LIN {X 0,Y 418.25,Z 348.011,A -85,B 0,C 180,E1 -10113.677,E2 -10113.677} C_VEL
LIN {X 0,Y 418.241,Z 348.013,A -85,B 0,C 180,E1 -10117.224,E2 -10117.224} C_VEL
LIN {X 0,Y 418.253,Z 348.011,A -85,B 0,C 180,E1 -10119.681,E2 -10119.681} C_VEL
LIN {X 0,Y 418.231,Z 348.014,A -85,B 0,C 180,E1 -10122.321,E2 -10122.321} C_VEL
LIN {X 0,Y 418.241,Z 348.014,A -85,B 0,C 180,E1 -10125.109,E2 -10125.109} C_VEL
LIN {X 0,Y 418.244,Z 348.011,A -85,B 0,C 180,E1 -10127.767,E2 -10127.767} C_VEL
LIN {X 0,Y 418.259,Z 348.01,A -85,B 0,C 180,E1 -10130.618,E2 -10130.618} C_VEL
LIN {X 0,Y 418.245,Z 348.013,A -85,B 0,C 180,E1 -10133.976,E2 -10133.976} C_VEL
LIN {X 0,Y 418.288,Z 348.13,A -85,B 0,C 180,E1 -10135.359,E2 -10135.359} C_VEL
LIN {X 0,Y 421.548,Z 360.205,A -85,B 0,C 180,E1 -10137.757,E2 -10137.757} C_VEL
LIN {X 0,Y 424.488,Z 372.309,A -85,B 0,C 180,E1 -10140.015,E2 -10140.015} C_VEL
LIN {X 0,Y 425.173,Z 376.878,A -85,B 0,C 180,E1 -10140.815,E2 -10140.815} C_VEL
LIN {X 0,Y 424.138,Z 389.684,A -85,B 0,C 180,E1 -10142.78,E2 -10142.78} C_VEL
LIN {X 0,Y 429.166,Z 416.83,A -85,B 0,C 180,E1 -10143.68,E2 -10143.68} C_VEL
LIN {X 0,Y 430.721,Z 426.232,A -85,B 0,C 180,E1 -10143.971,E2 -10143.971} C_VEL
LIN {X 0,Y 427.995,Z 557.544,A -85,B 0,C 180,E1 -10146.341,E2 -10146.341} C_VEL
LIN {X 0,Y 427.223,Z 573.369,A -85,B 0,C 180,E1 -10146.812,E2 -10146.812} C_VEL
LIN {X 0,Y 426.297,Z 587.688,A -85,B 0,C 180,E1 -10147.417,E2 -10147.417} C_VEL
LIN {X 0,Y 425.227,Z 601.253,A -85,B 0,C 180,E1 -10148.168,E2 -10148.168} C_VEL
LIN {X 0,Y 424.011,Z 614.986,A -85,B 0,C 180,E1 -10149.123,E2 -10149.123} C_VEL
LIN {X 0,Y 422.636,Z 628.963,A -85,B 0,C 180,E1 -10150.321,E2 -10150.321} C_VEL
LIN {X 0,Y 421.399,Z 641.731,A -85,B 0,C 180,E1 -10151.662,E2 -10151.662} C_VEL
LIN {X 0,Y 420.398,Z 652.28,A -85,B 0,C 180,E1 -10152.989,E2 -10152.989} C_VEL
LIN {X 0,Y 419.408,Z 662.178,A -85,B 0,C 180,E1 -10154.448,E2 -10154.448} C_VEL
LIN {X 0,Y 418.603,Z 671.918,A -85,B 0,C 180,E1 -10156.158,E2 -10156.158} C_VEL
LIN {X 0,Y 417.963,Z 680.043,A -85,B 0,C 180,E1 -10157.866,E2 -10157.866} C_VEL
LIN {X 0,Y 417.475,Z 687.641,A -85,B 0,C 180,E1 -10159.818,E2 -10159.818} C_VEL
LIN {X 0,Y 417.237,Z 693.683,A -85,B 0,C 180,E1 -10161.768,E2 -10161.768} C_VEL
LIN {X 0,Y 417.158,Z 698.338,A -85,B 0,C 180,E1 -10163.715,E2 -10163.715} C_VEL
LIN {X 0,Y 417.088,Z 700.928,A -85,B 0,C 180,E1 -10165.167,E2 -10165.167} C_VEL
LIN {X 0,Y 417.158,Z 703.338,A -85,B 0,C 180,E1 -10167.102,E2 -10167.102} C_VEL
LIN {X 0,Y 417.104,Z 704.552,A -85,B 0,C 180,E1 -10169.034,E2 -10169.034} C_VEL
LIN {X 0,Y 417.103,Z 704.581,A -85,B 0,C 180,E1 -10170.965,E2 -10170.965} C_VEL
LIN {X 0,Y 417.152,Z 703.387,A -85,B 0,C 180,E1 -10172.897,E2 -10172.897} C_VEL
LIN {X 0,Y 417.085,Z 700.995,A -85,B 0,C 180,E1 -10174.833,E2 -10174.833} C_VEL
LIN {X 0,Y 417.138,Z 697.366,A -85,B 0,C 180,E1 -10176.773,E2 -10176.773} C_VEL
LIN {X 0,Y 417.281,Z 692.404,A -85,B 0,C 180,E1 -10178.718,E2 -10178.718} C_VEL
LIN {X 0,Y 417.609,Z 685.98,A -85,B 0,C 180,E1 -10180.668,E2 -10180.668} C_VEL
LIN {X 0,Y 418.087,Z 677.912,A -85,B 0,C 180,E1 -10182.622,E2 -10182.622} C_VEL
LIN {X 0,Y 418.825,Z 669.323,A -85,B 0,C 180,E1 -10184.33,E2 -10184.33} C_VEL
LIN {X 0,Y 419.69,Z 658.966,A -85,B 0,C 180,E1 -10186.039,E2 -10186.039} C_VEL
LIN {X 0,Y 420.712,Z 648.387,A -85,B 0,C 180,E1 -10187.499,E2 -10187.499} C_VEL
LIN {X 0,Y 421.728,Z 636.884,A -85,B 0,C 180,E1 -10188.837,E2 -10188.837} C_VEL
LIN {X 0,Y 422.972,Z 624.401,A -85,B 0,C 180,E1 -10190.041,E2 -10190.041} C_VEL
LIN {X 0,Y 424.217,Z 610.764,A -85,B 0,C 180,E1 -10191.12,E2 -10191.12} C_VEL
LIN {X 0,Y 425.419,Z 596.688,A -85,B 0,C 180,E1 -10192.012,E2 -10192.012} C_VEL
LIN {X 0,Y 426.359,Z 582.366,A -85,B 0,C 180,E1 -10192.721,E2 -10192.721} C_VEL
LIN {X 0,Y 427.213,Z 566.762,A -85,B 0,C 180,E1 -10193.286,E2 -10193.286} C_VEL
LIN {X 0,Y 427.756,Z 550.147,A -85,B 0,C 180,E1 -10193.672,E2 -10193.672} C_VEL
LIN {X 0,Y 429.957,Z 432.408,A -85,B 0,C 180,E1 -10195.744,E2 -10195.744} C_VEL
LIN {X 0,Y 429.835,Z 424.529,A -85,B 0,C 180,E1 -10195.901,E2 -10195.901} C_VEL
LIN {X 0,Y 423.884,Z 391.337,A -85,B 0,C 180,E1 -10196.926,E2 -10196.926} C_VEL
LIN {X 0,Y 425.121,Z 376.572,A -85,B 0,C 180,E1 -10199.188,E2 -10199.188} C_VEL
LIN {X 0,Y 423.491,Z 368.485,A -85,B 0,C 180,E1 -10200.591,E2 -10200.591} C_VEL
LIN {X 0,Y 419.675,Z 353.216,A -85,B 0,C 180,E1 -10203.382,E2 -10203.382} C_VEL
LIN {X 0,Y 418.269,Z 348.009,A -85,B 0,C 180,E1 -10204.374,E2 -10204.374} C_VEL
LIN {X 0,Y 418.226,Z 348.018,A -85,B 0,C 180,E1 -10207.833,E2 -10207.833} C_VEL
LIN {X 0,Y 418.22,Z 348.014,A -85,B 0,C 180,E1 -10210.948,E2 -10210.948} C_VEL
LIN {X 0,Y 418.214,Z 348.013,A -85,B 0,C 180,E1 -10213.73,E2 -10213.73} C_VEL
LIN {X 0,Y 418.212,Z 348.012,A -85,B 0,C 180,E1 -10216.449,E2 -10216.449} C_VEL
LIN {X 0,Y 418.22,Z 348.017,A -85,B 0,C 180,E1 -10219.13,E2 -10219.13} C_VEL
LIN {X 0,Y 418.23,Z 348.009,A -85,B 0,C 180,E1 -10222.165,E2 -10222.165} C_VEL
LIN {X 0,Y 418.263,Z 348.009,A -85,B 0,C 180,E1 -10225.42,E2 -10225.42} C_VEL
LIN {X 0,Y 418.208,Z 348.014,A -85,B 0,C 180,E1 -10228.604,E2 -10228.604} C_VEL
LIN {X 0,Y 418.288,Z 348.002,A -85,B 0,C 180,E1 -10231.937,E2 -10231.937} C_VEL
LIN {X 0,Y 418.286,Z 348.009,A -85,B 0,C 180,E1 -10235.163,E2 -10235.163} C_VEL
LIN {X 0,Y 418.231,Z 348.01,A -85,B 0,C 180,E1 -10238.304,E2 -10238.304} C_VEL
LIN {X 0,Y 418.281,Z 348.006,A -85,B 0,C 180,E1 -10241.383,E2 -10241.383} C_VEL
LIN {X 0,Y 418.299,Z 348.002,A -85,B 0,C 180,E1 -10244.406,E2 -10244.406} C_VEL
LIN {X 0,Y 418.352,Z 347.997,A -85,B 0,C 180,E1 -10247.386,E2 -10247.386} C_VEL
LIN {X 0,Y 418.338,Z 347.997,A -85,B 0,C 180,E1 -10250.329,E2 -10250.329} C_VEL
LIN {X 0,Y 418.484,Z 347.981,A -85,B 0,C 180,E1 -10253.249,E2 -10253.249} C_VEL
LIN {X 0,Y 418.337,Z 348,A -85,B 0,C 180,E1 -10255.182,E2 -10255.182} C_VEL
LIN {X 0,Y 418.542,Z 347.97,A -85,B 0,C 180,E1 -10258.076,E2 -10258.076} C_VEL
LIN {X 0,Y 418.67,Z 347.954,A -85,B 0,C 180,E1 -10260,E2 -10260} C_VEL
LIN {X 0,Y 418.507,Z 347.982,A -85,B 0,C 180,E1 -10262.888,E2 -10262.888} C_VEL
LIN {X 0,Y 418.493,Z 347.983,A -85,B 0,C 180,E1 -10266.751,E2 -10266.751} C_VEL
LIN {X 0,Y 418.339,Z 347.996,A -85,B 0,C 180,E1 -10269.672,E2 -10269.672} C_VEL
LIN {X 0,Y 418.344,Z 348,A -85,B 0,C 180,E1 -10273.001,E2 -10273.001} C_VEL
LIN {X 0,Y 418.311,Z 348.006,A -85,B 0,C 180,E1 -10276.736,E2 -10276.736} C_VEL
LIN {X 0,Y 418.269,Z 348.004,A -85,B 0,C 180,E1 -10279.791,E2 -10279.791} C_VEL
LIN {X 0,Y 418.23,Z 348.017,A -85,B 0,C 180,E1 -10282.737,E2 -10282.737} C_VEL
LIN {X 0,Y 418.26,Z 348.006,A -85,B 0,C 180,E1 -10285.905,E2 -10285.905} C_VEL
LIN {X 0,Y 418.267,Z 348.007,A -85,B 0,C 180,E1 -10289.105,E2 -10289.105} C_VEL
LIN {X 0,Y 418.257,Z 348.011,A -85,B 0,C 180,E1 -10292.845,E2 -10292.845} C_VEL
LIN {X 0,Y 418.245,Z 348.01,A -85,B 0,C 180,E1 -10296.239,E2 -10296.239} C_VEL
LIN {X 0,Y 418.241,Z 348.008,A -85,B 0,C 180,E1 -10299.684,E2 -10299.684} C_VEL
LIN {X 0,Y 418.223,Z 348.014,A -85,B 0,C 180,E1 -10302.321,E2 -10302.321} C_VEL
LIN {X 0,Y 418.235,Z 348.01,A -85,B 0,C 180,E1 -10305.109,E2 -10305.109} C_VEL
LIN {X 0,Y 418.234,Z 348.009,A -85,B 0,C 180,E1 -10307.767,E2 -10307.767} C_VEL
LIN {X 0,Y 418.243,Z 348.014,A -85,B 0,C 180,E1 -10310.622,E2 -10310.622} C_VEL
LIN {X 0,Y 418.243,Z 348.009,A -85,B 0,C 180,E1 -10313.976,E2 -10313.976} C_VEL
LIN {X 0,Y 418.259,Z 348.006,A -85,B 0,C 180,E1 -10317.157,E2 -10317.157} C_VEL
LIN {X 0,Y 418.262,Z 348.008,A -85,B 0,C 180,E1 -10320.838,E2 -10320.838} C_VEL
LIN {X 0,Y 418.238,Z 348.011,A -85,B 0,C 180,E1 -10324.094,E2 -10324.094} C_VEL
LIN {X 0,Y 418.24,Z 348.008,A -85,B 0,C 180,E1 -10327.264,E2 -10327.264} C_VEL
LIN {X 0,Y 418.286,Z 348.009,A -85,B 0,C 180,E1 -10330.365,E2 -10330.365} C_VEL
LIN {X 0,Y 418.282,Z 348.003,A -85,B 0,C 180,E1 -10333.404,E2 -10333.404} C_VEL
LIN {X 0,Y 418.35,Z 347.995,A -85,B 0,C 180,E1 -10337,E2 -10337} C_VEL
LIN {X 0,Y 418.339,Z 348.003,A -85,B 0,C 180,E1 -10340.329,E2 -10340.329} C_VEL
LIN {X 0,Y 418.445,Z 347.982,A -85,B 0,C 180,E1 -10343.249,E2 -10343.249} C_VEL
LIN {X 0,Y 418.321,Z 347.998,A -85,B 0,C 180,E1 -10345.182,E2 -10345.182} C_VEL
LIN {X 0,Y 418.538,Z 347.976,A -85,B 0,C 180,E1 -10348.076,E2 -10348.076} C_VEL
LIN {X 0,Y 418.449,Z 347.983,A -85,B 0,C 180,E1 -10350.963,E2 -10350.963} C_VEL
LIN {X 0,Y 418.472,Z 347.98,A -85,B 0,C 180,E1 -10352.888,E2 -10352.888} C_VEL
LIN {X 0,Y 418.474,Z 347.981,A -85,B 0,C 180,E1 -10355.784,E2 -10355.784} C_VEL
LIN {X 0,Y 418.371,Z 347.994,A -85,B 0,C 180,E1 -10358.696,E2 -10358.696} C_VEL
LIN {X 0,Y 418.304,Z 348.002,A -85,B 0,C 180,E1 -10361.873,E2 -10361.873} C_VEL
LIN {X 0,Y 418.429,Z 348.896,A -85,B 0,C 180,E1 -10362.273,E2 -10362.273} C_VEL
LIN {X 0,Y 418.796,Z 351.663,A -85,B 0,C 180,E1 -10362.676,E2 -10362.676} C_VEL
LIN {X 0,Y 419.439,Z 356.854,A -85,B 0,C 180,E1 -10363.041,E2 -10363.041} C_VEL
LIN {X 0,Y 420.793,Z 367.676,A -85,B 0,C 180,E1 -10363.372,E2 -10363.372} C_VEL
LIN {X 0,Y 422.31,Z 374.12,A -85,B 0,C 180,E1 -10363.596,E2 -10363.596} C_VEL
LIN {X 0,Y 423.156,Z 376.108,A -85,B 0,C 180,E1 -10363.691,E2 -10363.691} C_VEL
LIN {X 0,Y 424.081,Z 378.351,A -85,B 0,C 180,E1 -10363.794,E2 -10363.794} C_VEL
LIN {X 0,Y 421.437,Z 512.397,A -85,B 0,C 180,E1 -10366.22,E2 -10366.22} C_VEL
LIN {X 0,Y 420.889,Z 527.525,A -85,B 0,C 180,E1 -10366.676,E2 -10366.676} C_VEL
LIN {X 0,Y 420.13,Z 542.435,A -85,B 0,C 180,E1 -10367.321,E2 -10367.321} C_VEL
LIN {X 0,Y 419.155,Z 556.684,A -85,B 0,C 180,E1 -10368.134,E2 -10368.134} C_VEL
LIN {X 0,Y 418.073,Z 570.507,A -85,B 0,C 180,E1 -10369.133,E2 -10369.133} C_VEL
LIN {X 0,Y 416.758,Z 584.238,A -85,B 0,C 180,E1 -10370.354,E2 -10370.354} C_VEL
LIN {X 0,Y 415.583,Z 596.693,A -85,B 0,C 180,E1 -10371.716,E2 -10371.716} C_VEL
LIN {X 0,Y 414.302,Z 608.449,A -85,B 0,C 180,E1 -10373.266,E2 -10373.266} C_VEL
LIN {X 0,Y 413.227,Z 618.693,A -85,B 0,C 180,E1 -10374.894,E2 -10374.894} C_VEL
LIN {X 0,Y 412.397,Z 627.476,A -85,B 0,C 180,E1 -10376.574,E2 -10376.574} C_VEL
LIN {X 0,Y 411.515,Z 636.067,A -85,B 0,C 180,E1 -10378.568,E2 -10378.568} C_VEL
LIN {X 0,Y 410.979,Z 642.087,A -85,B 0,C 180,E1 -10380.296,E2 -10380.296} C_VEL
LIN {X 0,Y 410.58,Z 647.031,A -85,B 0,C 180,E1 -10382.049,E2 -10382.049} C_VEL
LIN {X 0,Y 410.289,Z 650.99,A -85,B 0,C 180,E1 -10383.829,E2 -10383.829} C_VEL
LIN {X 0,Y 410.03,Z 653.979,A -85,B 0,C 180,E1 -10385.646,E2 -10385.646} C_VEL
LIN {X 0,Y 409.95,Z 655.413,A -85,B 0,C 180,E1 -10386.872,E2 -10386.872} C_VEL
LIN {X 0,Y 409.872,Z 656.387,A -85,B 0,C 180,E1 -10388.119,E2 -10388.119} C_VEL
LIN {X 0,Y 409.861,Z 656.932,A -85,B 0,C 180,E1 -10389.499,E2 -10389.499} C_VEL
LIN {X 0,Y 409.866,Z 656.925,A -85,B 0,C 180,E1 -10391.02,E2 -10391.02} C_VEL
LIN {X 0,Y 409.987,Z 655.627,A -85,B 0,C 180,E1 -10393.29,E2 -10393.29} C_VEL
LIN {X 0,Y 410.252,Z 653.041,A -85,B 0,C 180,E1 -10395.382,E2 -10395.382} C_VEL
LIN {X 0,Y 410.548,Z 649.25,A -85,B 0,C 180,E1 -10397.401,E2 -10397.401} C_VEL
LIN {X 0,Y 410.968,Z 643.973,A -85,B 0,C 180,E1 -10399.47,E2 -10399.47} C_VEL
LIN {X 0,Y 411.528,Z 637.967,A -85,B 0,C 180,E1 -10401.307,E2 -10401.307} C_VEL
LIN {X 0,Y 412.374,Z 630.184,A -85,B 0,C 180,E1 -10403.227,E2 -10403.227} C_VEL
LIN {X 0,Y 413.35,Z 621.249,A -85,B 0,C 180,E1 -10405.029,E2 -10405.029} C_VEL
LIN {X 0,Y 414.495,Z 611.153,A -85,B 0,C 180,E1 -10406.711,E2 -10406.711} C_VEL
LIN {X 0,Y 415.83,Z 599.954,A -85,B 0,C 180,E1 -10408.254,E2 -10408.254} C_VEL
LIN {X 0,Y 417.017,Z 588.013,A -85,B 0,C 180,E1 -10409.629,E2 -10409.629} C_VEL
LIN {X 0,Y 418.337,Z 574.777,A -85,B 0,C 180,E1 -10410.879,E2 -10410.879} C_VEL
LIN {X 0,Y 419.558,Z 561.572,A -85,B 0,C 180,E1 -10411.892,E2 -10411.892} C_VEL
LIN {X 0,Y 420.496,Z 548.182,A -85,B 0,C 180,E1 -10412.725,E2 -10412.725} C_VEL
LIN {X 0,Y 421.337,Z 533.466,A -85,B 0,C 180,E1 -10413.433,E2 -10413.433} C_VEL
LIN {X 0,Y 421.98,Z 518.146,A -85,B 0,C 180,E1 -10413.961,E2 -10413.961} C_VEL
LIN {X 0,Y 422.491,Z 497.901,A -85,B 0,C 180,E1 -10414.39,E2 -10414.39} C_VEL
LIN {X 0,Y 425.155,Z 379.31,A -85,B 0,C 180,E1 -10416.56,E2 -10416.56} C_VEL
LIN {X 0,Y 417.365,Z 362.024,A -85,B 0,C 180,E1 -10417.513,E2 -10417.513} C_VEL
LIN {X 0,Y 411.583,Z 350.448,A -85,B 0,C 180,E1 -10418.264,E2 -10418.264} C_VEL
LIN {X 0,Y 411.187,Z 348.889,A -85,B 0,C 180,E1 -10418.702,E2 -10418.702} C_VEL
LIN {X 0,Y 411.233,Z 348.884,A -85,B 0,C 180,E1 -10422.084,E2 -10422.084} C_VEL
LIN {X 0,Y 411.235,Z 348.885,A -85,B 0,C 180,E1 -10425.146,E2 -10425.146} C_VEL
LIN {X 0,Y 411.285,Z 348.88,A -85,B 0,C 180,E1 -10428.167,E2 -10428.167} C_VEL
LIN {X 0,Y 411.32,Z 348.873,A -85,B 0,C 180,E1 -10431.154,E2 -10431.154} C_VEL
LIN {X 0,Y 411.421,Z 348.861,A -85,B 0,C 180,E1 -10434.117,E2 -10434.117} C_VEL
LIN {X 0,Y 411.505,Z 348.852,A -85,B 0,C 180,E1 -10438.042,E2 -10438.042} C_VEL
LIN {X 0,Y 411.636,Z 348.836,A -85,B 0,C 180,E1 -10440,E2 -10440} C_VEL
LIN {X 0,Y 411.452,Z 348.856,A -85,B 0,C 180,E1 -10442.937,E2 -10442.937} C_VEL
LIN {X 0,Y 411.436,Z 348.86,A -85,B 0,C 180,E1 -10445.882,E2 -10445.882} C_VEL
LIN {X 0,Y 411.321,Z 348.874,A -85,B 0,C 180,E1 -10448.846,E2 -10448.846} C_VEL
LIN {X 0,Y 411.286,Z 348.877,A -85,B 0,C 180,E1 -10451.832,E2 -10451.832} C_VEL
LIN {X 0,Y 411.262,Z 348.881,A -85,B 0,C 180,E1 -10454.852,E2 -10454.852} C_VEL
LIN {X 0,Y 411.248,Z 348.879,A -85,B 0,C 180,E1 -10457.915,E2 -10457.915} C_VEL
LIN {X 0,Y 411.199,Z 348.888,A -85,B 0,C 180,E1 -10461.034,E2 -10461.034} C_VEL
LIN {X 0,Y 411.229,Z 348.88,A -85,B 0,C 180,E1 -10464.215,E2 -10464.215} C_VEL
LIN {X 0,Y 411.261,Z 348.88,A -85,B 0,C 180,E1 -10467.477,E2 -10467.477} C_VEL
LIN {X 0,Y 411.191,Z 348.89,A -85,B 0,C 180,E1 -10470.847,E2 -10470.847} C_VEL
LIN {X 0,Y 411.207,Z 348.888,A -85,B 0,C 180,E1 -10474.333,E2 -10474.333} C_VEL
LIN {X 0,Y 411.197,Z 348.89,A -85,B 0,C 180,E1 -10477.973,E2 -10477.973} C_VEL
LIN {X 0,Y 411.183,Z 348.893,A -85,B 0,C 180,E1 -10480.504,E2 -10480.504} C_VEL
LIN {X 0,Y 411.175,Z 348.893,A -85,B 0,C 180,E1 -10483.133,E2 -10483.133} C_VEL
LIN {X 0,Y 411.174,Z 348.892,A -85,B 0,C 180,E1 -10485.88,E2 -10485.88} C_VEL
LIN {X 0,Y 411.167,Z 348.897,A -85,B 0,C 180,E1 -10488.771,E2 -10488.771} C_VEL
LIN {X 0,Y 411.209,Z 348.89,A -85,B 0,C 180,E1 -10491.83,E2 -10491.83} C_VEL
LIN {X 0,Y 411.224,Z 348.94,A -85,B 0,C 180,E1 -10494.84,E2 -10494.84} C_VEL
LIN {X 0,Y 414.611,Z 361.305,A -85,B 0,C 180,E1 -10497.365,E2 -10497.365} C_VEL
LIN {X 0,Y 417.528,Z 373.326,A -85,B 0,C 180,E1 -10499.67,E2 -10499.67} C_VEL
LIN {X 0,Y 418.423,Z 378.327,A -85,B 0,C 180,E1 -10500.574,E2 -10500.574} C_VEL
LIN {X 0,Y 417.502,Z 389.145,A -85,B 0,C 180,E1 -10502.27,E2 -10502.27} C_VEL
LIN {X 0,Y 422.639,Z 416.531,A -85,B 0,C 180,E1 -10503.217,E2 -10503.217} C_VEL
LIN {X 0,Y 424.378,Z 426.949,A -85,B 0,C 180,E1 -10503.548,E2 -10503.548} C_VEL
LIN {X 0,Y 421.711,Z 550.656,A -85,B 0,C 180,E1 -10505.803,E2 -10505.803} C_VEL
LIN {X 0,Y 421.139,Z 566.163,A -85,B 0,C 180,E1 -10506.193,E2 -10506.193} C_VEL
LIN {X 0,Y 420.153,Z 581.384,A -85,B 0,C 180,E1 -10506.761,E2 -10506.761} C_VEL
LIN {X 0,Y 419.064,Z 596.003,A -85,B 0,C 180,E1 -10507.506,E2 -10507.506} C_VEL
LIN {X 0,Y 417.805,Z 609.905,A -85,B 0,C 180,E1 -10508.409,E2 -10508.409} C_VEL
LIN {X 0,Y 416.45,Z 623.415,A -85,B 0,C 180,E1 -10509.501,E2 -10509.501} C_VEL
LIN {X 0,Y 415.152,Z 635.852,A -85,B 0,C 180,E1 -10510.724,E2 -10510.724} C_VEL
LIN {X 0,Y 413.844,Z 648.291,A -85,B 0,C 180,E1 -10512.2,E2 -10512.2} C_VEL
LIN {X 0,Y 412.801,Z 658.729,A -85,B 0,C 180,E1 -10513.685,E2 -10513.685} C_VEL
LIN {X 0,Y 411.8,Z 668.967,A -85,B 0,C 180,E1 -10515.42,E2 -10515.42} C_VEL
LIN {X 0,Y 411.055,Z 677.485,A -85,B 0,C 180,E1 -10517.157,E2 -10517.157} C_VEL
LIN {X 0,Y 410.551,Z 685.519,A -85,B 0,C 180,E1 -10519.146,E2 -10519.146} C_VEL
LIN {X 0,Y 410.212,Z 691.921,A -85,B 0,C 180,E1 -10521.13,E2 -10521.13} C_VEL
LIN {X 0,Y 410.059,Z 696.883,A -85,B 0,C 180,E1 -10523.109,E2 -10523.109} C_VEL
LIN {X 0,Y 409.996,Z 700.525,A -85,B 0,C 180,E1 -10525.083,E2 -10525.083} C_VEL
LIN {X 0,Y 410.054,Z 702.931,A -85,B 0,C 180,E1 -10527.052,E2 -10527.052} C_VEL
LIN {X 0,Y 410.024,Z 704.142,A -85,B 0,C 180,E1 -10529.017,E2 -10529.017} C_VEL
LIN {X 0,Y 410.023,Z 704.169,A -85,B 0,C 180,E1 -10530.982,E2 -10530.982} C_VEL
LIN {X 0,Y 410.065,Z 702.966,A -85,B 0,C 180,E1 -10532.947,E2 -10532.947} C_VEL
LIN {X 0,Y 409.992,Z 700.562,A -85,B 0,C 180,E1 -10534.916,E2 -10534.916} C_VEL
LIN {X 0,Y 410.047,Z 696.919,A -85,B 0,C 180,E1 -10536.89,E2 -10536.89} C_VEL
LIN {X 0,Y 410.211,Z 691.942,A -85,B 0,C 180,E1 -10538.87,E2 -10538.87} C_VEL
LIN {X 0,Y 410.548,Z 685.5,A -85,B 0,C 180,E1 -10540.853,E2 -10540.853} C_VEL
LIN {X 0,Y 411.065,Z 677.411,A -85,B 0,C 180,E1 -10542.841,E2 -10542.841} C_VEL
LIN {X 0,Y 411.835,Z 668.798,A -85,B 0,C 180,E1 -10544.578,E2 -10544.578} C_VEL
LIN {X 0,Y 412.804,Z 658.417,A -85,B 0,C 180,E1 -10546.314,E2 -10546.314} C_VEL
LIN {X 0,Y 413.869,Z 647.806,A -85,B 0,C 180,E1 -10547.797,E2 -10547.797} C_VEL
LIN {X 0,Y 414.971,Z 636.266,A -85,B 0,C 180,E1 -10549.155,E2 -10549.155} C_VEL
LIN {X 0,Y 416.256,Z 623.742,A -85,B 0,C 180,E1 -10550.379,E2 -10550.379} C_VEL
LIN {X 0,Y 417.511,Z 610.038,A -85,B 0,C 180,E1 -10551.476,E2 -10551.476} C_VEL
LIN {X 0,Y 418.815,Z 595.894,A -85,B 0,C 180,E1 -10552.377,E2 -10552.377} C_VEL
LIN {X 0,Y 419.764,Z 581.088,A -85,B 0,C 180,E1 -10553.117,E2 -10553.117} C_VEL
LIN {X 0,Y 420.706,Z 565.62,A -85,B 0,C 180,E1 -10553.668,E2 -10553.668} C_VEL
LIN {X 0,Y 421.191,Z 550.165,A -85,B 0,C 180,E1 -10554.031,E2 -10554.031} C_VEL
LIN {X 0,Y 423.503,Z 432.336,A -85,B 0,C 180,E1 -10556.138,E2 -10556.138} C_VEL
LIN {X 0,Y 423.44,Z 426.12,A -85,B 0,C 180,E1 -10556.263,E2 -10556.263} C_VEL
LIN {X 0,Y 417.164,Z 390.938,A -85,B 0,C 180,E1 -10557.375,E2 -10557.375} C_VEL
LIN {X 0,Y 418.29,Z 377.717,A -85,B 0,C 180,E1 -10559.435,E2 -10559.435} C_VEL
LIN {X 0,Y 415.238,Z 364.235,A -85,B 0,C 180,E1 -10561.863,E2 -10561.863} C_VEL
LIN {X 0,Y 411.909,Z 351.557,A -85,B 0,C 180,E1 -10564.266,E2 -10564.266} C_VEL
LIN {X 0,Y 411.228,Z 348.889,A -85,B 0,C 180,E1 -10564.794,E2 -10564.794} C_VEL
LIN {X 0,Y 411.203,Z 348.893,A -85,B 0,C 180,E1 -10568.169,E2 -10568.169} C_VEL
LIN {X 0,Y 411.162,Z 348.897,A -85,B 0,C 180,E1 -10571.228,E2 -10571.228} C_VEL
LIN {X 0,Y 411.178,Z 348.888,A -85,B 0,C 180,E1 -10574.489,E2 -10574.489} C_VEL
LIN {X 0,Y 411.175,Z 348.888,A -85,B 0,C 180,E1 -10578.195,E2 -10578.195} C_VEL
LIN {X 0,Y 411.216,Z 348.886,A -85,B 0,C 180,E1 -10580.776,E2 -10580.776} C_VEL
LIN {X 0,Y 411.196,Z 348.886,A -85,B 0,C 180,E1 -10584.471,E2 -10584.471} C_VEL
LIN {X 0,Y 411.204,Z 348.889,A -85,B 0,C 180,E1 -10586.873,E2 -10586.873} C_VEL
LIN {X 0,Y 411.229,Z 348.883,A -85,B 0,C 180,E1 -10590.644,E2 -10590.644} C_VEL
LIN {X 0,Y 411.234,Z 348.882,A -85,B 0,C 180,E1 -10593.619,E2 -10593.619} C_VEL
LIN {X 0,Y 411.2,Z 348.89,A -85,B 0,C 180,E1 -10596.853,E2 -10596.853} C_VEL
LIN {X 0,Y 411.212,Z 348.883,A -85,B 0,C 180,E1 -10600.05,E2 -10600.05} C_VEL
LIN {X 0,Y 411.26,Z 348.884,A -85,B 0,C 180,E1 -10603.131,E2 -10603.131} C_VEL
LIN {X 0,Y 411.302,Z 348.878,A -85,B 0,C 180,E1 -10606.896,E2 -10606.896} C_VEL
LIN {X 0,Y 411.29,Z 348.874,A -85,B 0,C 180,E1 -10610.162,E2 -10610.162} C_VEL
LIN {X 0,Y 411.449,Z 348.859,A -85,B 0,C 180,E1 -10613.133,E2 -10613.133} C_VEL
LIN {X 0,Y 411.308,Z 348.877,A -85,B 0,C 180,E1 -10615.099,E2 -10615.099} C_VEL
LIN {X 0,Y 411.511,Z 348.846,A -85,B 0,C 180,E1 -10618.043,E2 -10618.043} C_VEL
LIN {X 0,Y 411.64,Z 348.83,A -85,B 0,C 180,E1 -10620,E2 -10620} C_VEL
LIN {X 0,Y 411.462,Z 348.859,A -85,B 0,C 180,E1 -10622.938,E2 -10622.938} C_VEL
LIN {X 0,Y 411.459,Z 348.86,A -85,B 0,C 180,E1 -10626.867,E2 -10626.867} C_VEL
LIN {X 0,Y 411.291,Z 348.874,A -85,B 0,C 180,E1 -10629.839,E2 -10629.839} C_VEL
LIN {X 0,Y 411.303,Z 348.876,A -85,B 0,C 180,E1 -10633.105,E2 -10633.105} C_VEL
LIN {X 0,Y 411.255,Z 348.884,A -85,B 0,C 180,E1 -10636.889,E2 -10636.889} C_VEL
LIN {X 0,Y 411.229,Z 348.882,A -85,B 0,C 180,E1 -10639.987,E2 -10639.987} C_VEL
LIN {X 0,Y 411.194,Z 348.888,A -85,B 0,C 180,E1 -10643.149,E2 -10643.149} C_VEL
LIN {X 0,Y 411.232,Z 348.884,A -85,B 0,C 180,E1 -10646.382,E2 -10646.382} C_VEL
LIN {X 0,Y 411.199,Z 348.885,A -85,B 0,C 180,E1 -10649.713,E2 -10649.713} C_VEL
LIN {X 0,Y 411.206,Z 348.886,A -85,B 0,C 180,E1 -10653.156,E2 -10653.156} C_VEL
LIN {X 0,Y 411.192,Z 348.892,A -85,B 0,C 180,E1 -10656.553,E2 -10656.553} C_VEL
LIN {X 0,Y 411.206,Z 348.884,A -85,B 0,C 180,E1 -10659.727,E2 -10659.727} C_VEL
LIN {X 0,Y 411.17,Z 348.89,A -85,B 0,C 180,E1 -10663.135,E2 -10663.135} C_VEL
LIN {X 0,Y 411.167,Z 348.89,A -85,B 0,C 180,E1 -10665.882,E2 -10665.882} C_VEL
LIN {X 0,Y 411.161,Z 348.894,A -85,B 0,C 180,E1 -10668.773,E2 -10668.773} C_VEL
LIN {X 0,Y 411.19,Z 348.888,A -85,B 0,C 180,E1 -10672.026,E2 -10672.026} C_VEL
LIN {X 0,Y 411.207,Z 348.884,A -85,B 0,C 180,E1 -10675.667,E2 -10675.667} C_VEL
LIN {X 0,Y 411.19,Z 348.887,A -85,B 0,C 180,E1 -10679.153,E2 -10679.153} C_VEL
LIN {X 0,Y 411.19,Z 348.893,A -85,B 0,C 180,E1 -10682.518,E2 -10682.518} C_VEL
LIN {X 0,Y 411.22,Z 348.883,A -85,B 0,C 180,E1 -10685.785,E2 -10685.785} C_VEL
LIN {X 0,Y 411.199,Z 348.887,A -85,B 0,C 180,E1 -10688.967,E2 -10688.967} C_VEL
LIN {X 0,Y 411.217,Z 348.886,A -85,B 0,C 180,E1 -10692.084,E2 -10692.084} C_VEL
LIN {X 0,Y 411.235,Z 348.881,A -85,B 0,C 180,E1 -10695.147,E2 -10695.147} C_VEL
LIN {X 0,Y 411.286,Z 348.879,A -85,B 0,C 180,E1 -10698.168,E2 -10698.168} C_VEL
LIN {X 0,Y 411.32,Z 348.87,A -85,B 0,C 180,E1 -10701.155,E2 -10701.155} C_VEL
LIN {X 0,Y 411.432,Z 348.861,A -85,B 0,C 180,E1 -10704.118,E2 -10704.118} C_VEL
LIN {X 0,Y 411.507,Z 348.851,A -85,B 0,C 180,E1 -10708.043,E2 -10708.043} C_VEL
LIN {X 0,Y 411.416,Z 348.859,A -85,B 0,C 180,E1 -10710.979,E2 -10710.979} C_VEL
LIN {X 0,Y 411.43,Z 348.857,A -85,B 0,C 180,E1 -10712.938,E2 -10712.938} C_VEL
LIN {X 0,Y 411.395,Z 348.866,A -85,B 0,C 180,E1 -10716.868,E2 -10716.868} C_VEL
LIN {X 0,Y 411.28,Z 348.878,A -85,B 0,C 180,E1 -10719.839,E2 -10719.839} C_VEL
LIN {X 0,Y 411.288,Z 348.878,A -85,B 0,C 180,E1 -10722.334,E2 -10722.334} C_VEL
LIN {X 0,Y 412.375,Z 351.826,A -85,B 0,C 180,E1 -10722.488,E2 -10722.488} C_VEL
LIN {X 0,Y 419.454,Z 367.142,A -85,B 0,C 180,E1 -10723.274,E2 -10723.274} C_VEL
LIN {X 0,Y 423.156,Z 376.108,A -85,B 0,C 180,E1 -10723.691,E2 -10723.691} C_VEL
LIN {X 0,Y 424.102,Z 379.628,A -85,B 0,C 180,E1 -10723.82,E2 -10723.82} C_VEL
LIN {X 0,Y 423.999,Z 383.414,A -85,B 0,C 180,E1 -10723.887,E2 -10723.887} C_VEL
LIN {X 0,Y 422.565,Z 389.18,A -85,B 0,C 180,E1 -10723.908,E2 -10723.908} C_VEL
LIN {X 0,Y 418.108,Z 400.97,A -85,B 0,C 180,E1 -10723.853,E2 -10723.853} C_VEL
LIN {X 0,Y 417.09,Z 406.1,A -85,B 0,C 180,E1 -10723.888,E2 -10723.888} C_VEL
LIN {X 0,Y 417.032,Z 407.139,A -85,B 0,C 180,E1 -10723.905,E2 -10723.905} C_VEL
LIN {X 0,Y 414.895,Z 512.721,A -85,B 0,C 180,E1 -10725.852,E2 -10725.852} C_VEL
LIN {X 0,Y 414.317,Z 527.935,A -85,B 0,C 180,E1 -10726.317,E2 -10726.317} C_VEL
LIN {X 0,Y 413.481,Z 543.381,A -85,B 0,C 180,E1 -10726.999,E2 -10726.999} C_VEL
LIN {X 0,Y 412.449,Z 558.069,A -85,B 0,C 180,E1 -10727.862,E2 -10727.862} C_VEL
LIN {X 0,Y 411.233,Z 572.569,A -85,B 0,C 180,E1 -10728.949,E2 -10728.949} C_VEL
LIN {X 0,Y 409.903,Z 585.924,A -85,B 0,C 180,E1 -10730.185,E2 -10730.185} C_VEL
LIN {X 0,Y 408.703,Z 597.748,A -85,B 0,C 180,E1 -10731.515,E2 -10731.515} C_VEL
LIN {X 0,Y 407.37,Z 609.522,A -85,B 0,C 180,E1 -10733.11,E2 -10733.11} C_VEL
LIN {X 0,Y 406.253,Z 619.872,A -85,B 0,C 180,E1 -10734.804,E2 -10734.804} C_VEL
LIN {X 0,Y 405.374,Z 628.572,A -85,B 0,C 180,E1 -10736.515,E2 -10736.515} C_VEL
LIN {X 0,Y 404.455,Z 637.028,A -85,B 0,C 180,E1 -10738.546,E2 -10738.546} C_VEL
LIN {X 0,Y 403.923,Z 642.992,A -85,B 0,C 180,E1 -10740.304,E2 -10740.304} C_VEL
LIN {X 0,Y 403.505,Z 647.832,A -85,B 0,C 180,E1 -10742.089,E2 -10742.089} C_VEL
LIN {X 0,Y 403.215,Z 651.685,A -85,B 0,C 180,E1 -10743.901,E2 -10743.901} C_VEL
LIN {X 0,Y 403.019,Z 653.718,A -85,B 0,C 180,E1 -10745.133,E2 -10745.133} C_VEL
LIN {X 0,Y 402.868,Z 655.609,A -85,B 0,C 180,E1 -10746.633,E2 -10746.633} C_VEL
LIN {X 0,Y 402.787,Z 657.205,A -85,B 0,C 180,E1 -10748.914,E2 -10748.914} C_VEL
LIN {X 0,Y 402.764,Z 657.446,A -85,B 0,C 180,E1 -10750.213,E2 -10750.213} C_VEL
LIN {X 0,Y 402.795,Z 657.18,A -85,B 0,C 180,E1 -10751.532,E2 -10751.532} C_VEL
LIN {X 0,Y 402.874,Z 656.404,A -85,B 0,C 180,E1 -10752.888,E2 -10752.888} C_VEL
LIN {X 0,Y 403.034,Z 654.99,A -85,B 0,C 180,E1 -10754.36,E2 -10754.36} C_VEL
LIN {X 0,Y 403.333,Z 651.839,A -85,B 0,C 180,E1 -10756.455,E2 -10756.455} C_VEL
LIN {X 0,Y 403.718,Z 647.256,A -85,B 0,C 180,E1 -10758.584,E2 -10758.584} C_VEL
LIN {X 0,Y 404.26,Z 641.471,A -85,B 0,C 180,E1 -10760.613,E2 -10760.613} C_VEL
LIN {X 0,Y 405.059,Z 634.266,A -85,B 0,C 180,E1 -10762.607,E2 -10762.607} C_VEL
LIN {X 0,Y 406.03,Z 626.084,A -85,B 0,C 180,E1 -10764.443,E2 -10764.443} C_VEL
LIN {X 0,Y 407.139,Z 616.398,A -85,B 0,C 180,E1 -10766.237,E2 -10766.237} C_VEL
LIN {X 0,Y 408.497,Z 605.399,A -85,B 0,C 180,E1 -10767.914,E2 -10767.914} C_VEL
LIN {X 0,Y 409.824,Z 593.954,A -85,B 0,C 180,E1 -10769.364,E2 -10769.364} C_VEL
LIN {X 0,Y 411.143,Z 581.575,A -85,B 0,C 180,E1 -10770.667,E2 -10770.667} C_VEL
LIN {X 0,Y 412.493,Z 568.233,A -85,B 0,C 180,E1 -10771.816,E2 -10771.816} C_VEL
LIN {X 0,Y 413.54,Z 554.746,A -85,B 0,C 180,E1 -10772.761,E2 -10772.761} C_VEL
LIN {X 0,Y 414.61,Z 539.998,A -85,B 0,C 180,E1 -10773.563,E2 -10773.563} C_VEL
LIN {X 0,Y 415.324,Z 524.735,A -85,B 0,C 180,E1 -10774.184,E2 -10774.184} C_VEL
LIN {X 0,Y 415.877,Z 509.671,A -85,B 0,C 180,E1 -10774.59,E2 -10774.59} C_VEL
LIN {X 0,Y 418.807,Z 380.978,A -85,B 0,C 180,E1 -10777.005,E2 -10777.005} C_VEL
LIN {X 0,Y 411.068,Z 364.109,A -85,B 0,C 180,E1 -10777.978,E2 -10777.978} C_VEL
LIN {X 0,Y 404.428,Z 351.022,A -85,B 0,C 180,E1 -10778.863,E2 -10778.863} C_VEL
LIN {X 0,Y 404.158,Z 349.765,A -85,B 0,C 180,E1 -10779.182,E2 -10779.182} C_VEL
LIN {X 0,Y 404.184,Z 349.758,A -85,B 0,C 180,E1 -10782.806,E2 -10782.806} C_VEL
LIN {X 0,Y 404.27,Z 349.753,A -85,B 0,C 180,E1 -10786.788,E2 -10786.788} C_VEL
LIN {X 0,Y 404.257,Z 349.756,A -85,B 0,C 180,E1 -10789.988,E2 -10789.988} C_VEL
LIN {X 0,Y 404.344,Z 349.742,A -85,B 0,C 180,E1 -10793.011,E2 -10793.011} C_VEL
LIN {X 0,Y 404.262,Z 349.752,A -85,B 0,C 180,E1 -10795.013,E2 -10795.013} C_VEL
LIN {X 0,Y 404.474,Z 349.728,A -85,B 0,C 180,E1 -10798.008,E2 -10798.008} C_VEL
LIN {X 0,Y 404.606,Z 349.711,A -85,B 0,C 180,E1 -10800,E2 -10800} C_VEL
LIN {X 0,Y 404.41,Z 349.734,A -85,B 0,C 180,E1 -10802.988,E2 -10802.988} C_VEL
LIN {X 0,Y 404.384,Z 349.738,A -85,B 0,C 180,E1 -10805.985,E2 -10805.985} C_VEL
LIN {X 0,Y 404.268,Z 349.754,A -85,B 0,C 180,E1 -10809.001,E2 -10809.001} C_VEL
LIN {X 0,Y 404.258,Z 349.751,A -85,B 0,C 180,E1 -10812.041,E2 -10812.041} C_VEL
LIN {X 0,Y 404.208,Z 349.759,A -85,B 0,C 180,E1 -10815.118,E2 -10815.118} C_VEL
LIN {X 0,Y 404.207,Z 349.755,A -85,B 0,C 180,E1 -10818.238,E2 -10818.238} C_VEL
LIN {X 0,Y 404.141,Z 349.765,A -85,B 0,C 180,E1 -10821.419,E2 -10821.419} C_VEL
LIN {X 0,Y 404.179,Z 349.759,A -85,B 0,C 180,E1 -10824.665,E2 -10824.665} C_VEL
LIN {X 0,Y 404.197,Z 349.76,A -85,B 0,C 180,E1 -10827.999,E2 -10827.999} C_VEL
LIN {X 0,Y 404.141,Z 349.767,A -85,B 0,C 180,E1 -10831.558,E2 -10831.558} C_VEL
LIN {X 0,Y 404.186,Z 349.763,A -85,B 0,C 180,E1 -10835.016,E2 -10835.016} C_VEL
LIN {X 0,Y 404.157,Z 349.769,A -85,B 0,C 180,E1 -10838.756,E2 -10838.756} C_VEL
LIN {X 0,Y 404.124,Z 349.772,A -85,B 0,C 180,E1 -10841.599,E2 -10841.599} C_VEL
LIN {X 0,Y 404.148,Z 349.769,A -85,B 0,C 180,E1 -10844.522,E2 -10844.522} C_VEL
LIN {X 0,Y 404.141,Z 349.77,A -85,B 0,C 180,E1 -10847.296,E2 -10847.296} C_VEL
LIN {X 0,Y 404.17,Z 349.768,A -85,B 0,C 180,E1 -10849.955,E2 -10849.955} C_VEL
LIN {X 0,Y 404.138,Z 349.767,A -85,B 0,C 180,E1 -10853.124,E2 -10853.124} C_VEL
LIN {X 0,Y 404.194,Z 349.94,A -85,B 0,C 180,E1 -10854.332,E2 -10854.332} C_VEL
LIN {X 0,Y 407.891,Z 363.192,A -85,B 0,C 180,E1 -10857.121,E2 -10857.121} C_VEL
LIN {X 0,Y 410.719,Z 374.785,A -85,B 0,C 180,E1 -10859.398,E2 -10859.398} C_VEL
LIN {X 0,Y 411.649,Z 379.776,A -85,B 0,C 180,E1 -10860.322,E2 -10860.322} C_VEL
LIN {X 0,Y 410.963,Z 388.779,A -85,B 0,C 180,E1 -10861.746,E2 -10861.746} C_VEL
LIN {X 0,Y 415.839,Z 414.516,A -85,B 0,C 180,E1 -10862.67,E2 -10862.67} C_VEL
LIN {X 0,Y 418.094,Z 428.387,A -85,B 0,C 180,E1 -10863.126,E2 -10863.126} C_VEL
LIN {X 0,Y 415.159,Z 555.509,A -85,B 0,C 180,E1 -10865.496,E2 -10865.496} C_VEL
LIN {X 0,Y 414.376,Z 571.677,A -85,B 0,C 180,E1 -10865.98,E2 -10865.98} C_VEL
LIN {X 0,Y 413.363,Z 585.751,A -85,B 0,C 180,E1 -10866.583,E2 -10866.583} C_VEL
LIN {X 0,Y 412.179,Z 598.93,A -85,B 0,C 180,E1 -10867.315,E2 -10867.315} C_VEL
LIN {X 0,Y 410.868,Z 612.837,A -85,B 0,C 180,E1 -10868.29,E2 -10868.29} C_VEL
LIN {X 0,Y 409.474,Z 625.714,A -85,B 0,C 180,E1 -10869.399,E2 -10869.399} C_VEL
LIN {X 0,Y 408.005,Z 638.783,A -85,B 0,C 180,E1 -10870.765,E2 -10870.765} C_VEL
LIN {X 0,Y 406.819,Z 649.757,A -85,B 0,C 180,E1 -10872.143,E2 -10872.143} C_VEL
LIN {X 0,Y 405.742,Z 659.928,A -85,B 0,C 180,E1 -10873.651,E2 -10873.651} C_VEL
LIN {X 0,Y 404.73,Z 669.894,A -85,B 0,C 180,E1 -10875.416,E2 -10875.416} C_VEL
LIN {X 0,Y 403.968,Z 677.964,A -85,B 0,C 180,E1 -10877.12,E2 -10877.12} C_VEL
LIN {X 0,Y 403.503,Z 685.134,A -85,B 0,C 180,E1 -10878.954,E2 -10878.954} C_VEL
LIN {X 0,Y 403.134,Z 691.525,A -85,B 0,C 180,E1 -10880.973,E2 -10880.973} C_VEL
LIN {X 0,Y 402.981,Z 696.485,A -85,B 0,C 180,E1 -10882.987,E2 -10882.987} C_VEL
LIN {X 0,Y 402.908,Z 700.125,A -85,B 0,C 180,E1 -10884.996,E2 -10884.996} C_VEL
LIN {X 0,Y 402.952,Z 702.526,A -85,B 0,C 180,E1 -10887,E2 -10887} C_VEL
LIN {X 0,Y 402.946,Z 703.733,A -85,B 0,C 180,E1 -10889,E2 -10889} C_VEL
LIN {X 0,Y 402.946,Z 703.756,A -85,B 0,C 180,E1 -10890.999,E2 -10890.999} C_VEL
LIN {X 0,Y 402.962,Z 702.544,A -85,B 0,C 180,E1 -10892.999,E2 -10892.999} C_VEL
LIN {X 0,Y 402.902,Z 700.13,A -85,B 0,C 180,E1 -10895.003,E2 -10895.003} C_VEL
LIN {X 0,Y 402.968,Z 696.474,A -85,B 0,C 180,E1 -10897.012,E2 -10897.012} C_VEL
LIN {X 0,Y 403.133,Z 691.48,A -85,B 0,C 180,E1 -10899.027,E2 -10899.027} C_VEL
LIN {X 0,Y 403.501,Z 685.02,A -85,B 0,C 180,E1 -10901.045,E2 -10901.045} C_VEL
LIN {X 0,Y 404.07,Z 676.912,A -85,B 0,C 180,E1 -10903.068,E2 -10903.068} C_VEL
LIN {X 0,Y 404.877,Z 668.274,A -85,B 0,C 180,E1 -10904.834,E2 -10904.834} C_VEL
LIN {X 0,Y 405.927,Z 657.868,A -85,B 0,C 180,E1 -10906.599,E2 -10906.599} C_VEL
LIN {X 0,Y 407.027,Z 647.211,A -85,B 0,C 180,E1 -10908.107,E2 -10908.107} C_VEL
LIN {X 0,Y 408.186,Z 635.615,A -85,B 0,C 180,E1 -10909.486,E2 -10909.486} C_VEL
LIN {X 0,Y 409.536,Z 623.02,A -85,B 0,C 180,E1 -10910.728,E2 -10910.728} C_VEL
LIN {X 0,Y 410.863,Z 609.223,A -85,B 0,C 180,E1 -10911.841,E2 -10911.841} C_VEL
LIN {X 0,Y 412.191,Z 594.769,A -85,B 0,C 180,E1 -10912.767,E2 -10912.767} C_VEL
LIN {X 0,Y 413.191,Z 579.944,A -85,B 0,C 180,E1 -10913.507,E2 -10913.507} C_VEL
LIN {X 0,Y 414.126,Z 565.227,A -85,B 0,C 180,E1 -10914.035,E2 -10914.035} C_VEL
LIN {X 0,Y 414.642,Z 549.798,A -85,B 0,C 180,E1 -10914.402,E2 -10914.402} C_VEL
LIN {X 0,Y 417.041,Z 431.156,A -85,B 0,C 180,E1 -10916.563,E2 -10916.563} C_VEL
LIN {X 0,Y 416.91,Z 426.848,A -85,B 0,C 180,E1 -10916.656,E2 -10916.656} C_VEL
LIN {X 0,Y 410.507,Z 390.685,A -85,B 0,C 180,E1 -10917.809,E2 -10917.809} C_VEL
LIN {X 0,Y 411.446,Z 380.579,A -85,B 0,C 180,E1 -10919.409,E2 -10919.409} C_VEL
LIN {X 0,Y 411.019,Z 377.12,A -85,B 0,C 180,E1 -10920.009,E2 -10920.009} C_VEL
LIN {X 0,Y 407.922,Z 364.127,A -85,B 0,C 180,E1 -10922.413,E2 -10922.413} C_VEL
LIN {X 0,Y 404.695,Z 351.832,A -85,B 0,C 180,E1 -10924.799,E2 -10924.799} C_VEL
LIN {X 0,Y 404.165,Z 349.765,A -85,B 0,C 180,E1 -10925.24,E2 -10925.24} C_VEL
LIN {X 0,Y 404.153,Z 349.773,A -85,B 0,C 180,E1 -10928.756,E2 -10928.756} C_VEL
LIN {X 0,Y 404.122,Z 349.77,A -85,B 0,C 180,E1 -10931.6,E2 -10931.6} C_VEL
LIN {X 0,Y 404.147,Z 349.764,A -85,B 0,C 180,E1 -10934.523,E2 -10934.523} C_VEL
LIN {X 0,Y 404.136,Z 349.771,A -85,B 0,C 180,E1 -10937.296,E2 -10937.296} C_VEL
LIN {X 0,Y 404.165,Z 349.762,A -85,B 0,C 180,E1 -10939.955,E2 -10939.955} C_VEL
LIN {X 0,Y 404.136,Z 349.772,A -85,B 0,C 180,E1 -10943.124,E2 -10943.124} C_VEL
LIN {X 0,Y 404.142,Z 349.764,A -85,B 0,C 180,E1 -10946.188,E2 -10946.188} C_VEL
LIN {X 0,Y 404.142,Z 349.765,A -85,B 0,C 180,E1 -10949.715,E2 -10949.715} C_VEL
LIN {X 0,Y 404.192,Z 349.765,A -85,B 0,C 180,E1 -10953.123,E2 -10953.123} C_VEL
LIN {X 0,Y 404.174,Z 349.764,A -85,B 0,C 180,E1 -10955.334,E2 -10955.334} C_VEL
LIN {X 0,Y 404.135,Z 349.767,A -85,B 0,C 180,E1 -10958.581,E2 -10958.581} C_VEL
LIN {X 0,Y 404.207,Z 349.757,A -85,B 0,C 180,E1 -10961.762,E2 -10961.762} C_VEL
LIN {X 0,Y 404.204,Z 349.762,A -85,B 0,C 180,E1 -10964.882,E2 -10964.882} C_VEL
LIN {X 0,Y 404.254,Z 349.75,A -85,B 0,C 180,E1 -10967.959,E2 -10967.959} C_VEL
LIN {X 0,Y 404.402,Z 349.732,A -85,B 0,C 180,E1 -10972.129,E2 -10972.129} C_VEL
LIN {X 0,Y 404.416,Z 349.73,A -85,B 0,C 180,E1 -10974.015,E2 -10974.015} C_VEL
LIN {X 0,Y 404.48,Z 349.722,A -85,B 0,C 180,E1 -10978.009,E2 -10978.009} C_VEL
LIN {X 0,Y 404.609,Z 349.706,A -85,B 0,C 180,E1 -10980,E2 -10980} C_VEL
LIN {X 0,Y 404.419,Z 349.736,A -85,B 0,C 180,E1 -10982.989,E2 -10982.989} C_VEL
LIN {X 0,Y 404.41,Z 349.736,A -85,B 0,C 180,E1 -10986.988,E2 -10986.988} C_VEL
LIN {X 0,Y 404.256,Z 349.75,A -85,B 0,C 180,E1 -10990.012,E2 -10990.012} C_VEL
LIN {X 0,Y 404.264,Z 349.752,A -85,B 0,C 180,E1 -10993.212,E2 -10993.212} C_VEL
LIN {X 0,Y 404.214,Z 349.76,A -85,B 0,C 180,E1 -10997.008,E2 -10997.008} C_VEL
LIN {X 0,Y 404.162,Z 349.764,A -85,B 0,C 180,E1 -11000.352,E2 -11000.352} C_VEL
LIN {X 0,Y 404.159,Z 349.762,A -85,B 0,C 180,E1 -11003.576,E2 -11003.576} C_VEL
LIN {X 0,Y 404.18,Z 349.759,A -85,B 0,C 180,E1 -11005.767,E2 -11005.767} C_VEL
LIN {X 0,Y 404.194,Z 349.758,A -85,B 0,C 180,E1 -11008,E2 -11008} C_VEL
LIN {X 0,Y 404.138,Z 349.765,A -85,B 0,C 180,E1 -11011.559,E2 -11011.559} C_VEL
LIN {X 0,Y 404.184,Z 349.762,A -85,B 0,C 180,E1 -11015.017,E2 -11015.017} C_VEL
LIN {X 0,Y 404.148,Z 349.769,A -85,B 0,C 180,E1 -11018.758,E2 -11018.758} C_VEL
LIN {X 0,Y 404.118,Z 349.767,A -85,B 0,C 180,E1 -11021.6,E2 -11021.6} C_VEL
LIN {X 0,Y 404.145,Z 349.77,A -85,B 0,C 180,E1 -11024.523,E2 -11024.523} C_VEL
LIN {X 0,Y 404.133,Z 349.766,A -85,B 0,C 180,E1 -11027.296,E2 -11027.296} C_VEL
LIN {X 0,Y 404.154,Z 349.764,A -85,B 0,C 180,E1 -11029.954,E2 -11029.954} C_VEL
LIN {X 0,Y 404.136,Z 349.766,A -85,B 0,C 180,E1 -11033.126,E2 -11033.126} C_VEL
LIN {X 0,Y 404.146,Z 349.767,A -85,B 0,C 180,E1 -11036.188,E2 -11036.188} C_VEL
LIN {X 0,Y 404.146,Z 349.764,A -85,B 0,C 180,E1 -11039.715,E2 -11039.715} C_VEL
LIN {X 0,Y 404.136,Z 349.766,A -85,B 0,C 180,E1 -11043.119,E2 -11043.119} C_VEL
LIN {X 0,Y 404.168,Z 349.768,A -85,B 0,C 180,E1 -11046.426,E2 -11046.426} C_VEL
LIN {X 0,Y 404.194,Z 349.759,A -85,B 0,C 180,E1 -11049.875,E2 -11049.875} C_VEL
LIN {X 0,Y 404.177,Z 349.761,A -85,B 0,C 180,E1 -11053.013,E2 -11053.013} C_VEL
LIN {X 0,Y 404.286,Z 349.747,A -85,B 0,C 180,E1 -11056.939,E2 -11056.939} C_VEL
LIN {X 0,Y 404.258,Z 349.753,A -85,B 0,C 180,E1 -11059.989,E2 -11059.989} C_VEL
LIN {X 0,Y 404.344,Z 349.74,A -85,B 0,C 180,E1 -11063.012,E2 -11063.012} C_VEL
LIN {X 0,Y 404.265,Z 349.749,A -85,B 0,C 180,E1 -11065.014,E2 -11065.014} C_VEL
LIN {X 0,Y 404.475,Z 349.727,A -85,B 0,C 180,E1 -11068.009,E2 -11068.009} C_VEL
LIN {X 0,Y 404.383,Z 349.735,A -85,B 0,C 180,E1 -11070.996,E2 -11070.996} C_VEL
LIN {X 0,Y 404.39,Z 349.734,A -85,B 0,C 180,E1 -11072.989,E2 -11072.989} C_VEL
LIN {X 0,Y 404.371,Z 349.74,A -85,B 0,C 180,E1 -11075.986,E2 -11075.986} C_VEL
LIN {X 0,Y 404.26,Z 349.75,A -85,B 0,C 180,E1 -11079.002,E2 -11079.002} C_VEL
LIN {X 0,Y 404.231,Z 349.759,A -85,B 0,C 180,E1 -11081.852,E2 -11081.852} C_VEL
LIN {X 0,Y 405.34,Z 352.724,A -85,B 0,C 180,E1 -11082.009,E2 -11082.009} C_VEL
LIN {X 0,Y 412.959,Z 368.878,A -85,B 0,C 180,E1 -11082.873,E2 -11082.873} C_VEL
LIN {X 0,Y 417.601,Z 380.024,A -85,B 0,C 180,E1 -11083.407,E2 -11083.407} C_VEL
LIN {X 0,Y 417.032,Z 407.139,A -85,B 0,C 180,E1 -11083.905,E2 -11083.905} C_VEL
LIN {X 0,Y 416.28,Z 412.982,A -85,B 0,C 180,E1 -11083.971,E2 -11083.971} C_VEL
LIN {X 0,Y 410.636,Z 432.001,A -85,B 0,C 180,E1 -11083.985,E2 -11083.985} C_VEL
LIN {X 0,Y 409.9,Z 437.842,A -85,B 0,C 180,E1 -11084.055,E2 -11084.055} C_VEL
LIN {X 0,Y 408.332,Z 513.825,A -85,B 0,C 180,E1 -11085.491,E2 -11085.491} C_VEL
LIN {X 0,Y 407.749,Z 528.828,A -85,B 0,C 180,E1 -11085.965,E2 -11085.965} C_VEL
LIN {X 0,Y 406.913,Z 543.483,A -85,B 0,C 180,E1 -11086.623,E2 -11086.623} C_VEL
LIN {X 0,Y 405.916,Z 557.118,A -85,B 0,C 180,E1 -11087.426,E2 -11087.426} C_VEL
LIN {X 0,Y 404.733,Z 571.27,A -85,B 0,C 180,E1 -11088.476,E2 -11088.476} C_VEL
LIN {X 0,Y 403.272,Z 585.297,A -85,B 0,C 180,E1 -11089.764,E2 -11089.764} C_VEL
LIN {X 0,Y 401.983,Z 597.463,A -85,B 0,C 180,E1 -11091.137,E2 -11091.137} C_VEL
LIN {X 0,Y 400.671,Z 608.972,A -85,B 0,C 180,E1 -11092.7,E2 -11092.7} C_VEL
LIN {X 0,Y 399.465,Z 619.489,A -85,B 0,C 180,E1 -11094.421,E2 -11094.421} C_VEL
LIN {X 0,Y 398.498,Z 628.315,A -85,B 0,C 180,E1 -11096.162,E2 -11096.162} C_VEL
LIN {X 0,Y 397.525,Z 636.714,A -85,B 0,C 180,E1 -11098.171,E2 -11098.171} C_VEL
LIN {X 0,Y 396.861,Z 643.88,A -85,B 0,C 180,E1 -11100.327,E2 -11100.327} C_VEL
LIN {X 0,Y 396.434,Z 648.614,A -85,B 0,C 180,E1 -11102.13,E2 -11102.13} C_VEL
LIN {X 0,Y 396.194,Z 651.558,A -85,B 0,C 180,E1 -11103.516,E2 -11103.516} C_VEL
LIN {X 0,Y 395.924,Z 654.395,A -85,B 0,C 180,E1 -11105.259,E2 -11105.259} C_VEL
LIN {X 0,Y 395.737,Z 656.507,A -85,B 0,C 180,E1 -11107.144,E2 -11107.144} C_VEL
LIN {X 0,Y 395.693,Z 657.457,A -85,B 0,C 180,E1 -11108.601,E2 -11108.601} C_VEL
LIN {X 0,Y 395.7,Z 657.861,A -85,B 0,C 180,E1 -11110.206,E2 -11110.206} C_VEL
LIN {X 0,Y 395.751,Z 657.207,A -85,B 0,C 180,E1 -11112.441,E2 -11112.441} C_VEL
LIN {X 0,Y 396.013,Z 655.033,A -85,B 0,C 180,E1 -11114.775,E2 -11114.775} C_VEL
LIN {X 0,Y 396.303,Z 652.166,A -85,B 0,C 180,E1 -11116.643,E2 -11116.643} C_VEL
LIN {X 0,Y 396.662,Z 648.094,A -85,B 0,C 180,E1 -11118.58,E2 -11118.58} C_VEL
LIN {X 0,Y 397.157,Z 643.103,A -85,B 0,C 180,E1 -11120.427,E2 -11120.427} C_VEL
LIN {X 0,Y 397.851,Z 637.018,A -85,B 0,C 180,E1 -11122.246,E2 -11122.246} C_VEL
LIN {X 0,Y 398.819,Z 629.155,A -85,B 0,C 180,E1 -11124.157,E2 -11124.157} C_VEL
LIN {X 0,Y 399.824,Z 621.14,A -85,B 0,C 180,E1 -11125.771,E2 -11125.771} C_VEL
LIN {X 0,Y 400.964,Z 612.28,A -85,B 0,C 180,E1 -11127.282,E2 -11127.282} C_VEL
LIN {X 0,Y 402.369,Z 601.305,A -85,B 0,C 180,E1 -11128.856,E2 -11128.856} C_VEL
LIN {X 0,Y 403.65,Z 589.861,A -85,B 0,C 180,E1 -11130.231,E2 -11130.231} C_VEL
LIN {X 0,Y 405.059,Z 577.068,A -85,B 0,C 180,E1 -11131.501,E2 -11131.501} C_VEL
LIN {X 0,Y 406.445,Z 563.59,A -85,B 0,C 180,E1 -11132.588,E2 -11132.588} C_VEL
LIN {X 0,Y 407.509,Z 550.199,A -85,B 0,C 180,E1 -11133.462,E2 -11133.462} C_VEL
LIN {X 0,Y 408.433,Z 535.931,A -85,B 0,C 180,E1 -11134.186,E2 -11134.186} C_VEL
LIN {X 0,Y 409.145,Z 520.619,A -85,B 0,C 180,E1 -11134.753,E2 -11134.753} C_VEL
LIN {X 0,Y 409.69,Z 504.851,A -85,B 0,C 180,E1 -11135.125,E2 -11135.125} C_VEL
LIN {X 0,Y 412.673,Z 383.294,A -85,B 0,C 180,E1 -11137.435,E2 -11137.435} C_VEL
LIN {X 0,Y 405.842,Z 368.219,A -85,B 0,C 180,E1 -11138.327,E2 -11138.327} C_VEL
LIN {X 0,Y 398.596,Z 354.223,A -85,B 0,C 180,E1 -11139.283,E2 -11139.283} C_VEL
LIN {X 0,Y 397.307,Z 351.544,A -85,B 0,C 180,E1 -11139.495,E2 -11139.495} C_VEL
LIN {X 0,Y 397.125,Z 350.645,A -85,B 0,C 180,E1 -11139.771,E2 -11139.771} C_VEL
LIN {X 0,Y 397.157,Z 350.633,A -85,B 0,C 180,E1 -11142.858,E2 -11142.858} C_VEL
LIN {X 0,Y 397.232,Z 350.63,A -85,B 0,C 180,E1 -11146.702,E2 -11146.702} C_VEL
LIN {X 0,Y 397.217,Z 350.633,A -85,B 0,C 180,E1 -11149.809,E2 -11149.809} C_VEL
LIN {X 0,Y 397.296,Z 350.619,A -85,B 0,C 180,E1 -11152.887,E2 -11152.887} C_VEL
LIN {X 0,Y 397.233,Z 350.627,A -85,B 0,C 180,E1 -11154.924,E2 -11154.924} C_VEL
LIN {X 0,Y 397.443,Z 350.604,A -85,B 0,C 180,E1 -11157.973,E2 -11157.973} C_VEL
LIN {X 0,Y 397.575,Z 350.587,A -85,B 0,C 180,E1 -11160,E2 -11160} C_VEL
LIN {X 0,Y 397.369,Z 350.611,A -85,B 0,C 180,E1 -11163.041,E2 -11163.041} C_VEL
LIN {X 0,Y 397.335,Z 350.615,A -85,B 0,C 180,E1 -11166.092,E2 -11166.092} C_VEL
LIN {X 0,Y 397.238,Z 350.63,A -85,B 0,C 180,E1 -11169.162,E2 -11169.162} C_VEL
LIN {X 0,Y 397.222,Z 350.627,A -85,B 0,C 180,E1 -11172.258,E2 -11172.258} C_VEL
LIN {X 0,Y 397.181,Z 350.632,A -85,B 0,C 180,E1 -11175.392,E2 -11175.392} C_VEL
LIN {X 0,Y 397.16,Z 350.633,A -85,B 0,C 180,E1 -11178.573,E2 -11178.573} C_VEL
LIN {X 0,Y 397.099,Z 350.643,A -85,B 0,C 180,E1 -11181.818,E2 -11181.818} C_VEL
LIN {X 0,Y 397.159,Z 350.637,A -85,B 0,C 180,E1 -11185.131,E2 -11185.131} C_VEL
LIN {X 0,Y 397.164,Z 350.637,A -85,B 0,C 180,E1 -11187.776,E2 -11187.776} C_VEL
LIN {X 0,Y 397.081,Z 350.648,A -85,B 0,C 180,E1 -11190.882,E2 -11190.882} C_VEL
LIN {X 0,Y 397.127,Z 350.643,A -85,B 0,C 180,E1 -11194.493,E2 -11194.493} C_VEL
LIN {X 0,Y 397.105,Z 350.646,A -85,B 0,C 180,E1 -11198.274,E2 -11198.274} C_VEL
LIN {X 0,Y 397.09,Z 350.648,A -85,B 0,C 180,E1 -11200.908,E2 -11200.908} C_VEL
LIN {X 0,Y 397.102,Z 350.646,A -85,B 0,C 180,E1 -11203.648,E2 -11203.648} C_VEL
LIN {X 0,Y 397.106,Z 350.645,A -85,B 0,C 180,E1 -11206.52,E2 -11206.52} C_VEL
LIN {X 0,Y 397.115,Z 350.644,A -85,B 0,C 180,E1 -11210.423,E2 -11210.423} C_VEL
LIN {X 0,Y 397.141,Z 350.769,A -85,B 0,C 180,E1 -11213.759,E2 -11213.759} C_VEL
LIN {X 0,Y 401.118,Z 364.77,A -85,B 0,C 180,E1 -11216.802,E2 -11216.802} C_VEL
LIN {X 0,Y 404.266,Z 378.09,A -85,B 0,C 180,E1 -11219.463,E2 -11219.463} C_VEL
LIN {X 0,Y 404.932,Z 382.026,A -85,B 0,C 180,E1 -11220.203,E2 -11220.203} C_VEL
LIN {X 0,Y 404.375,Z 387.873,A -85,B 0,C 180,E1 -11221.172,E2 -11221.172} C_VEL
LIN {X 0,Y 409.259,Z 413.431,A -85,B 0,C 180,E1 -11222.139,E2 -11222.139} C_VEL
LIN {X 0,Y 411.833,Z 429.86,A -85,B 0,C 180,E1 -11222.686,E2 -11222.686} C_VEL
LIN {X 0,Y 408.719,Z 555.947,A -85,B 0,C 180,E1 -11225.084,E2 -11225.084} C_VEL
LIN {X 0,Y 407.904,Z 571.736,A -85,B 0,C 180,E1 -11225.574,E2 -11225.574} C_VEL
LIN {X 0,Y 406.784,Z 586.666,A -85,B 0,C 180,E1 -11226.233,E2 -11226.233} C_VEL
LIN {X 0,Y 405.397,Z 601.294,A -85,B 0,C 180,E1 -11227.085,E2 -11227.085} C_VEL
LIN {X 0,Y 403.915,Z 615.761,A -85,B 0,C 180,E1 -11228.166,E2 -11228.166} C_VEL
LIN {X 0,Y 402.299,Z 629.314,A -85,B 0,C 180,E1 -11229.416,E2 -11229.416} C_VEL
LIN {X 0,Y 400.877,Z 641.7,A -85,B 0,C 180,E1 -11230.809,E2 -11230.809} C_VEL
LIN {X 0,Y 399.62,Z 653.038,A -85,B 0,C 180,E1 -11232.339,E2 -11232.339} C_VEL
LIN {X 0,Y 398.353,Z 664.077,A -85,B 0,C 180,E1 -11234.129,E2 -11234.129} C_VEL
LIN {X 0,Y 397.415,Z 673.301,A -85,B 0,C 180,E1 -11235.927,E2 -11235.927} C_VEL
LIN {X 0,Y 396.737,Z 680.973,A -85,B 0,C 180,E1 -11237.726,E2 -11237.726} C_VEL
LIN {X 0,Y 396.182,Z 688.14,A -85,B 0,C 180,E1 -11239.782,E2 -11239.782} C_VEL
LIN {X 0,Y 395.958,Z 693.791,A -85,B 0,C 180,E1 -11241.836,E2 -11241.836} C_VEL
LIN {X 0,Y 395.859,Z 698.072,A -85,B 0,C 180,E1 -11243.885,E2 -11243.885} C_VEL
LIN {X 0,Y 395.788,Z 701.075,A -85,B 0,C 180,E1 -11245.927,E2 -11245.927} C_VEL
LIN {X 0,Y 395.916,Z 702.874,A -85,B 0,C 180,E1 -11247.965,E2 -11247.965} C_VEL
LIN {X 0,Y 395.871,Z 703.485,A -85,B 0,C 180,E1 -11250,E2 -11250} C_VEL
LIN {X 0,Y 395.914,Z 702.886,A -85,B 0,C 180,E1 -11252.034,E2 -11252.034} C_VEL
LIN {X 0,Y 395.786,Z 701.06,A -85,B 0,C 180,E1 -11254.073,E2 -11254.073} C_VEL
LIN {X 0,Y 395.857,Z 697.933,A -85,B 0,C 180,E1 -11256.166,E2 -11256.166} C_VEL
LIN {X 0,Y 395.948,Z 693.697,A -85,B 0,C 180,E1 -11258.163,E2 -11258.163} C_VEL
LIN {X 0,Y 396.181,Z 687.964,A -85,B 0,C 180,E1 -11260.218,E2 -11260.218} C_VEL
LIN {X 0,Y 396.774,Z 680.687,A -85,B 0,C 180,E1 -11262.272,E2 -11262.272} C_VEL
LIN {X 0,Y 397.427,Z 672.885,A -85,B 0,C 180,E1 -11264.072,E2 -11264.072} C_VEL
LIN {X 0,Y 398.325,Z 663.493,A -85,B 0,C 180,E1 -11265.871,E2 -11265.871} C_VEL
LIN {X 0,Y 399.452,Z 653.952,A -85,B 0,C 180,E1 -11267.403,E2 -11267.403} C_VEL
LIN {X 0,Y 400.657,Z 641.864,A -85,B 0,C 180,E1 -11269.028,E2 -11269.028} C_VEL
LIN {X 0,Y 402.035,Z 628.883,A -85,B 0,C 180,E1 -11270.464,E2 -11270.464} C_VEL
LIN {X 0,Y 403.402,Z 616.475,A -85,B 0,C 180,E1 -11271.594,E2 -11271.594} C_VEL
LIN {X 0,Y 404.884,Z 601.733,A -85,B 0,C 180,E1 -11272.677,E2 -11272.677} C_VEL
LIN {X 0,Y 406.081,Z 587.081,A -85,B 0,C 180,E1 -11273.524,E2 -11273.524} C_VEL
LIN {X 0,Y 407.105,Z 572.152,A -85,B 0,C 180,E1 -11274.171,E2 -11274.171} C_VEL
LIN {X 0,Y 407.854,Z 556.824,A -85,B 0,C 180,E1 -11274.632,E2 -11274.632} C_VEL
LIN {X 0,Y 410.583,Z 433.685,A -85,B 0,C 180,E1 -11276.928,E2 -11276.928} C_VEL
LIN {X 0,Y 410.545,Z 428.307,A -85,B 0,C 180,E1 -11277.038,E2 -11277.038} C_VEL
LIN {X 0,Y 403.869,Z 390.135,A -85,B 0,C 180,E1 -11278.306,E2 -11278.306} C_VEL
LIN {X 0,Y 404.635,Z 381.354,A -85,B 0,C 180,E1 -11279.723,E2 -11279.723} C_VEL
LIN {X 0,Y 402.085,Z 369.635,A -85,B 0,C 180,E1 -11281.897,E2 -11281.897} C_VEL
LIN {X 0,Y 398.492,Z 355.846,A -85,B 0,C 180,E1 -11284.595,E2 -11284.595} C_VEL
LIN {X 0,Y 397.119,Z 350.643,A -85,B 0,C 180,E1 -11285.654,E2 -11285.654} C_VEL
LIN {X 0,Y 397.111,Z 350.644,A -85,B 0,C 180,E1 -11289.577,E2 -11289.577} C_VEL
LIN {X 0,Y 397.102,Z 350.645,A -85,B 0,C 180,E1 -11293.479,E2 -11293.479} C_VEL
LIN {X 0,Y 397.102,Z 350.642,A -85,B 0,C 180,E1 -11296.52,E2 -11296.52} C_VEL
LIN {X 0,Y 397.111,Z 350.641,A -85,B 0,C 180,E1 -11300.423,E2 -11300.423} C_VEL
LIN {X 0,Y 397.106,Z 350.641,A -85,B 0,C 180,E1 -11304.265,E2 -11304.265} C_VEL
LIN {X 0,Y 397.111,Z 350.643,A -85,B 0,C 180,E1 -11306.727,E2 -11306.727} C_VEL
LIN {X 0,Y 397.121,Z 350.639,A -85,B 0,C 180,E1 -11310.296,E2 -11310.296} C_VEL
LIN {X 0,Y 397.191,Z 350.632,A -85,B 0,C 180,E1 -11312.61,E2 -11312.61} C_VEL
LIN {X 0,Y 397.13,Z 350.638,A -85,B 0,C 180,E1 -11315.982,E2 -11315.982} C_VEL
LIN {X 0,Y 397.135,Z 350.638,A -85,B 0,C 180,E1 -11319.705,E2 -11319.705} C_VEL
LIN {X 0,Y 397.178,Z 350.637,A -85,B 0,C 180,E1 -11322.845,E2 -11322.845} C_VEL
LIN {X 0,Y 397.225,Z 350.629,A -85,B 0,C 180,E1 -11326.703,E2 -11326.703} C_VEL
LIN {X 0,Y 397.215,Z 350.627,A -85,B 0,C 180,E1 -11329.809,E2 -11329.809} C_VEL
LIN {X 0,Y 397.347,Z 350.617,A -85,B 0,C 180,E1 -11332.888,E2 -11332.888} C_VEL
LIN {X 0,Y 397.251,Z 350.63,A -85,B 0,C 180,E1 -11334.925,E2 -11334.925} C_VEL
LIN {X 0,Y 397.449,Z 350.598,A -85,B 0,C 180,E1 -11337.974,E2 -11337.974} C_VEL
LIN {X 0,Y 397.578,Z 350.582,A -85,B 0,C 180,E1 -11340,E2 -11340} C_VEL
LIN {X 0,Y 397.378,Z 350.612,A -85,B 0,C 180,E1 -11343.042,E2 -11343.042} C_VEL
LIN {X 0,Y 397.362,Z 350.613,A -85,B 0,C 180,E1 -11347.112,E2 -11347.112} C_VEL
LIN {X 0,Y 397.216,Z 350.628,A -85,B 0,C 180,E1 -11350.191,E2 -11350.191} C_VEL
LIN {X 0,Y 397.224,Z 350.628,A -85,B 0,C 180,E1 -11353.322,E2 -11353.322} C_VEL
LIN {X 0,Y 397.18,Z 350.634,A -85,B 0,C 180,E1 -11357.156,E2 -11357.156} C_VEL
LIN {X 0,Y 397.101,Z 350.648,A -85,B 0,C 180,E1 -11360.731,E2 -11360.731} C_VEL
LIN {X 0,Y 397.124,Z 350.639,A -85,B 0,C 180,E1 -11364.019,E2 -11364.019} C_VEL
LIN {X 0,Y 397.192,Z 350.631,A -85,B 0,C 180,E1 -11367.391,E2 -11367.391} C_VEL
LIN {X 0,Y 397.078,Z 350.649,A -85,B 0,C 180,E1 -11370.883,E2 -11370.883} C_VEL
LIN {X 0,Y 397.125,Z 350.643,A -85,B 0,C 180,E1 -11374.494,E2 -11374.494} C_VEL
LIN {X 0,Y 397.098,Z 350.645,A -85,B 0,C 180,E1 -11378.276,E2 -11378.276} C_VEL
LIN {X 0,Y 397.086,Z 350.647,A -85,B 0,C 180,E1 -11380.91,E2 -11380.91} C_VEL
LIN {X 0,Y 397.1,Z 350.641,A -85,B 0,C 180,E1 -11383.649,E2 -11383.649} C_VEL
LIN {X 0,Y 397.101,Z 350.648,A -85,B 0,C 180,E1 -11386.522,E2 -11386.522} C_VEL
LIN {X 0,Y 397.103,Z 350.647,A -85,B 0,C 180,E1 -11390.422,E2 -11390.422} C_VEL
LIN {X 0,Y 397.109,Z 350.645,A -85,B 0,C 180,E1 -11394.266,E2 -11394.266} C_VEL
LIN {X 0,Y 397.116,Z 350.644,A -85,B 0,C 180,E1 -11396.728,E2 -11396.728} C_VEL
LIN {X 0,Y 397.12,Z 350.644,A -85,B 0,C 180,E1 -11400.296,E2 -11400.296} C_VEL
LIN {X 0,Y 397.097,Z 350.642,A -85,B 0,C 180,E1 -11403.74,E2 -11403.74} C_VEL
LIN {X 0,Y 397.11,Z 350.641,A -85,B 0,C 180,E1 -11407.086,E2 -11407.086} C_VEL
LIN {X 0,Y 397.148,Z 350.642,A -85,B 0,C 180,E1 -11410.353,E2 -11410.353} C_VEL
LIN {X 0,Y 397.131,Z 350.638,A -85,B 0,C 180,E1 -11413.552,E2 -11413.552} C_VEL
LIN {X 0,Y 397.232,Z 350.628,A -85,B 0,C 180,E1 -11416.703,E2 -11416.703} C_VEL
LIN {X 0,Y 397.218,Z 350.628,A -85,B 0,C 180,E1 -11419.809,E2 -11419.809} C_VEL
LIN {X 0,Y 397.297,Z 350.618,A -85,B 0,C 180,E1 -11422.887,E2 -11422.887} C_VEL
LIN {X 0,Y 397.236,Z 350.625,A -85,B 0,C 180,E1 -11424.925,E2 -11424.925} C_VEL
LIN {X 0,Y 397.444,Z 350.602,A -85,B 0,C 180,E1 -11427.974,E2 -11427.974} C_VEL
LIN {X 0,Y 397.443,Z 350.603,A -85,B 0,C 180,E1 -11432.027,E2 -11432.027} C_VEL
LIN {X 0,Y 397.324,Z 350.619,A -85,B 0,C 180,E1 -11436.093,E2 -11436.093} C_VEL
LIN {X 0,Y 397.231,Z 350.625,A -85,B 0,C 180,E1 -11439.163,E2 -11439.163} C_VEL
LIN {X 0,Y 397.206,Z 350.63,A -85,B 0,C 180,E1 -11441.366,E2 -11441.366} C_VEL
LIN {X 0,Y 398.248,Z 353.569,A -85,B 0,C 180,E1 -11441.513,E2 -11441.513} C_VEL
LIN {X 0,Y 405.554,Z 368.544,A -85,B 0,C 180,E1 -11442.352,E2 -11442.352} C_VEL
LIN {X 0,Y 411.162,Z 381.942,A -85,B 0,C 180,E1 -11443.015,E2 -11443.015} C_VEL
LIN {X 0,Y 409.9,Z 437.842,A -85,B 0,C 180,E1 -11444.055,E2 -11444.055} C_VEL
LIN {X 0,Y 409.141,Z 443.689,A -85,B 0,C 180,E1 -11444.123,E2 -11444.123} C_VEL
LIN {X 0,Y 403.421,Z 462.7,A -85,B 0,C 180,E1 -11444.135,E2 -11444.135} C_VEL
LIN {X 0,Y 402.766,Z 468.541,A -85,B 0,C 180,E1 -11444.21,E2 -11444.21} C_VEL
LIN {X 0,Y 401.782,Z 514.699,A -85,B 0,C 180,E1 -11445.114,E2 -11445.114} C_VEL
LIN {X 0,Y 401.147,Z 529.974,A -85,B 0,C 180,E1 -11445.613,E2 -11445.613} C_VEL
LIN {X 0,Y 400.236,Z 545.111,A -85,B 0,C 180,E1 -11446.318,E2 -11446.318} C_VEL
LIN {X 0,Y 399.195,Z 558.817,A -85,B 0,C 180,E1 -11447.151,E2 -11447.151} C_VEL
LIN {X 0,Y 398.032,Z 572.087,A -85,B 0,C 180,E1 -11448.166,E2 -11448.166} C_VEL
LIN {X 0,Y 396.593,Z 585.368,A -85,B 0,C 180,E1 -11449.407,E2 -11449.407} C_VEL
LIN {X 0,Y 395.201,Z 597.861,A -85,B 0,C 180,E1 -11450.835,E2 -11450.835} C_VEL
LIN {X 0,Y 393.854,Z 609.268,A -85,B 0,C 180,E1 -11452.408,E2 -11452.408} C_VEL
LIN {X 0,Y 392.642,Z 619.451,A -85,B 0,C 180,E1 -11454.095,E2 -11454.095} C_VEL
LIN {X 0,Y 391.622,Z 628.134,A -85,B 0,C 180,E1 -11455.821,E2 -11455.821} C_VEL
LIN {X 0,Y 390.742,Z 635.579,A -85,B 0,C 180,E1 -11457.591,E2 -11457.591} C_VEL
LIN {X 0,Y 389.977,Z 642.505,A -85,B 0,C 180,E1 -11459.594,E2 -11459.594} C_VEL
LIN {X 0,Y 389.492,Z 647.906,A -85,B 0,C 180,E1 -11461.553,E2 -11461.553} C_VEL
LIN {X 0,Y 389.072,Z 652.621,A -85,B 0,C 180,E1 -11463.806,E2 -11463.806} C_VEL
LIN {X 0,Y 388.792,Z 655.32,A -85,B 0,C 180,E1 -11465.565,E2 -11465.565} C_VEL
LIN {X 0,Y 388.639,Z 657.546,A -85,B 0,C 180,E1 -11467.941,E2 -11467.941} C_VEL
LIN {X 0,Y 388.594,Z 658.118,A -85,B 0,C 180,E1 -11469.272,E2 -11469.272} C_VEL
LIN {X 0,Y 388.616,Z 658.225,A -85,B 0,C 180,E1 -11470.621,E2 -11470.621} C_VEL
LIN {X 0,Y 388.656,Z 657.788,A -85,B 0,C 180,E1 -11472.149,E2 -11472.149} C_VEL
LIN {X 0,Y 388.763,Z 656.737,A -85,B 0,C 180,E1 -11473.687,E2 -11473.687} C_VEL
LIN {X 0,Y 388.99,Z 655.019,A -85,B 0,C 180,E1 -11475.2,E2 -11475.2} C_VEL
LIN {X 0,Y 389.232,Z 652.769,A -85,B 0,C 180,E1 -11476.675,E2 -11476.675} C_VEL
LIN {X 0,Y 389.641,Z 648.598,A -85,B 0,C 180,E1 -11478.718,E2 -11478.718} C_VEL
LIN {X 0,Y 390.257,Z 642.647,A -85,B 0,C 180,E1 -11480.927,E2 -11480.927} C_VEL
LIN {X 0,Y 391.148,Z 635.531,A -85,B 0,C 180,E1 -11482.992,E2 -11482.992} C_VEL
LIN {X 0,Y 392.325,Z 626.829,A -85,B 0,C 180,E1 -11485.023,E2 -11485.023} C_VEL
LIN {X 0,Y 393.465,Z 617.916,A -85,B 0,C 180,E1 -11486.739,E2 -11486.739} C_VEL
LIN {X 0,Y 394.941,Z 607.148,A -85,B 0,C 180,E1 -11488.458,E2 -11488.458} C_VEL
LIN {X 0,Y 396.374,Z 595.986,A -85,B 0,C 180,E1 -11489.941,E2 -11489.941} C_VEL
LIN {X 0,Y 397.754,Z 584.507,A -85,B 0,C 180,E1 -11491.217,E2 -11491.217} C_VEL
LIN {X 0,Y 399.156,Z 572.345,A -85,B 0,C 180,E1 -11492.342,E2 -11492.342} C_VEL
LIN {X 0,Y 400.408,Z 558.779,A -85,B 0,C 180,E1 -11493.374,E2 -11493.374} C_VEL
LIN {X 0,Y 401.491,Z 545.1,A -85,B 0,C 180,E1 -11494.201,E2 -11494.201} C_VEL
LIN {X 0,Y 402.422,Z 529.939,A -85,B 0,C 180,E1 -11494.893,E2 -11494.893} C_VEL
LIN {X 0,Y 403.063,Z 514.787,A -85,B 0,C 180,E1 -11495.376,E2 -11495.376} C_VEL
LIN {X 0,Y 406.436,Z 385.1,A -85,B 0,C 180,E1 -11497.905,E2 -11497.905} C_VEL
LIN {X 0,Y 398.811,Z 368.54,A -85,B 0,C 180,E1 -11498.939,E2 -11498.939} C_VEL
LIN {X 0,Y 391.718,Z 355.211,A -85,B 0,C 180,E1 -11499.904,E2 -11499.904} C_VEL
LIN {X 0,Y 390.344,Z 352.666,A -85,B 0,C 180,E1 -11500.098,E2 -11500.098} C_VEL
LIN {X 0,Y 390.222,Z 352.233,A -85,B 0,C 180,E1 -11500.126,E2 -11500.126} C_VEL
LIN {X 0,Y 390.088,Z 351.516,A -85,B 0,C 180,E1 -11500.393,E2 -11500.393} C_VEL
LIN {X 0,Y 390.109,Z 351.512,A -85,B 0,C 180,E1 -11503.247,E2 -11503.247} C_VEL
LIN {X 0,Y 390.198,Z 351.507,A -85,B 0,C 180,E1 -11506.561,E2 -11506.561} C_VEL
LIN {X 0,Y 390.169,Z 351.509,A -85,B 0,C 180,E1 -11509.622,E2 -11509.622} C_VEL
LIN {X 0,Y 390.249,Z 351.497,A -85,B 0,C 180,E1 -11512.757,E2 -11512.757} C_VEL
LIN {X 0,Y 390.204,Z 351.503,A -85,B 0,C 180,E1 -11514.833,E2 -11514.833} C_VEL
LIN {X 0,Y 390.41,Z 351.481,A -85,B 0,C 180,E1 -11517.936,E2 -11517.936} C_VEL
LIN {X 0,Y 390.545,Z 351.462,A -85,B 0,C 180,E1 -11520,E2 -11520} C_VEL
LIN {X 0,Y 390.304,Z 351.492,A -85,B 0,C 180,E1 -11523.096,E2 -11523.096} C_VEL
LIN {X 0,Y 390.288,Z 351.492,A -85,B 0,C 180,E1 -11526.202,E2 -11526.202} C_VEL
LIN {X 0,Y 390.195,Z 351.505,A -85,B 0,C 180,E1 -11529.329,E2 -11529.329} C_VEL
LIN {X 0,Y 390.173,Z 351.505,A -85,B 0,C 180,E1 -11532.483,E2 -11532.483} C_VEL
LIN {X 0,Y 390.141,Z 351.507,A -85,B 0,C 180,E1 -11535.676,E2 -11535.676} C_VEL
LIN {X 0,Y 390.105,Z 351.512,A -85,B 0,C 180,E1 -11538.922,E2 -11538.922} C_VEL
LIN {X 0,Y 390.042,Z 351.522,A -85,B 0,C 180,E1 -11542.234,E2 -11542.234} C_VEL
LIN {X 0,Y 390.121,Z 351.515,A -85,B 0,C 180,E1 -11545.743,E2 -11545.743} C_VEL
LIN {X 0,Y 390.061,Z 351.522,A -85,B 0,C 180,E1 -11549.109,E2 -11549.109} C_VEL
LIN {X 0,Y 390.044,Z 351.522,A -85,B 0,C 180,E1 -11552.721,E2 -11552.721} C_VEL
LIN {X 0,Y 390.057,Z 351.524,A -85,B 0,C 180,E1 -11555.825,E2 -11555.825} C_VEL
LIN {X 0,Y 390.071,Z 351.522,A -85,B 0,C 180,E1 -11559.218,E2 -11559.218} C_VEL
LIN {X 0,Y 390.044,Z 351.526,A -85,B 0,C 180,E1 -11562.374,E2 -11562.374} C_VEL
LIN {X 0,Y 390.048,Z 351.526,A -85,B 0,C 180,E1 -11565.354,E2 -11565.354} C_VEL
LIN {X 0,Y 390.034,Z 351.527,A -85,B 0,C 180,E1 -11568.187,E2 -11568.187} C_VEL
LIN {X 0,Y 390.092,Z 351.516,A -85,B 0,C 180,E1 -11570.907,E2 -11570.907} C_VEL
LIN {X 0,Y 390.08,Z 351.61,A -85,B 0,C 180,E1 -11573.157,E2 -11573.157} C_VEL
LIN {X 0,Y 393.938,Z 365.023,A -85,B 0,C 180,E1 -11576.175,E2 -11576.175} C_VEL
LIN {X 0,Y 397.193,Z 378.326,A -85,B 0,C 180,E1 -11578.928,E2 -11578.928} C_VEL
LIN {X 0,Y 398.189,Z 384.431,A -85,B 0,C 180,E1 -11580.101,E2 -11580.101} C_VEL
LIN {X 0,Y 397.913,Z 387.621,A -85,B 0,C 180,E1 -11580.616,E2 -11580.616} C_VEL
LIN {X 0,Y 402.6,Z 411.83,A -85,B 0,C 180,E1 -11581.563,E2 -11581.563} C_VEL
LIN {X 0,Y 405.601,Z 430.52,A -85,B 0,C 180,E1 -11582.215,E2 -11582.215} C_VEL
LIN {X 0,Y 402.377,Z 555.266,A -85,B 0,C 180,E1 -11584.629,E2 -11584.629} C_VEL
LIN {X 0,Y 401.512,Z 571.085,A -85,B 0,C 180,E1 -11585.125,E2 -11585.125} C_VEL
LIN {X 0,Y 400.376,Z 585.687,A -85,B 0,C 180,E1 -11585.776,E2 -11585.776} C_VEL
LIN {X 0,Y 398.942,Z 600,A -85,B 0,C 180,E1 -11586.611,E2 -11586.611} C_VEL
LIN {X 0,Y 397.485,Z 614.029,A -85,B 0,C 180,E1 -11587.657,E2 -11587.657} C_VEL
LIN {X 0,Y 395.795,Z 627.839,A -85,B 0,C 180,E1 -11588.926,E2 -11588.926} C_VEL
LIN {X 0,Y 394.213,Z 640.391,A -85,B 0,C 180,E1 -11590.336,E2 -11590.336} C_VEL
LIN {X 0,Y 392.764,Z 652.857,A -85,B 0,C 180,E1 -11592.041,E2 -11592.041} C_VEL
LIN {X 0,Y 391.439,Z 663.742,A -85,B 0,C 180,E1 -11593.841,E2 -11593.841} C_VEL
LIN {X 0,Y 390.45,Z 672.939,A -85,B 0,C 180,E1 -11595.67,E2 -11595.67} C_VEL
LIN {X 0,Y 389.709,Z 680.602,A -85,B 0,C 180,E1 -11597.501,E2 -11597.501} C_VEL
LIN {X 0,Y 389.129,Z 687.764,A -85,B 0,C 180,E1 -11599.594,E2 -11599.594} C_VEL
LIN {X 0,Y 388.888,Z 693.41,A -85,B 0,C 180,E1 -11601.687,E2 -11601.687} C_VEL
LIN {X 0,Y 388.794,Z 697.779,A -85,B 0,C 180,E1 -11603.825,E2 -11603.825} C_VEL
LIN {X 0,Y 388.709,Z 700.679,A -85,B 0,C 180,E1 -11605.852,E2 -11605.852} C_VEL
LIN {X 0,Y 388.845,Z 702.47,A -85,B 0,C 180,E1 -11607.928,E2 -11607.928} C_VEL
LIN {X 0,Y 388.796,Z 703.071,A -85,B 0,C 180,E1 -11610,E2 -11610} C_VEL
LIN {X 0,Y 388.845,Z 702.468,A -85,B 0,C 180,E1 -11612.071,E2 -11612.071} C_VEL
LIN {X 0,Y 388.708,Z 700.626,A -85,B 0,C 180,E1 -11614.147,E2 -11614.147} C_VEL
LIN {X 0,Y 388.773,Z 697.574,A -85,B 0,C 180,E1 -11616.226,E2 -11616.226} C_VEL
LIN {X 0,Y 388.881,Z 693.225,A -85,B 0,C 180,E1 -11618.312,E2 -11618.312} C_VEL
LIN {X 0,Y 389.127,Z 687.468,A -85,B 0,C 180,E1 -11620.405,E2 -11620.405} C_VEL
LIN {X 0,Y 389.738,Z 680.164,A -85,B 0,C 180,E1 -11622.497,E2 -11622.497} C_VEL
LIN {X 0,Y 390.454,Z 672.335,A -85,B 0,C 180,E1 -11624.329,E2 -11624.329} C_VEL
LIN {X 0,Y 391.37,Z 662.906,A -85,B 0,C 180,E1 -11626.161,E2 -11626.161} C_VEL
LIN {X 0,Y 392.568,Z 653.336,A -85,B 0,C 180,E1 -11627.718,E2 -11627.718} C_VEL
LIN {X 0,Y 393.771,Z 641.943,A -85,B 0,C 180,E1 -11629.28,E2 -11629.28} C_VEL
LIN {X 0,Y 395.158,Z 629.452,A -85,B 0,C 180,E1 -11630.7,E2 -11630.7} C_VEL
LIN {X 0,Y 396.746,Z 615.686,A -85,B 0,C 180,E1 -11631.975,E2 -11631.975} C_VEL
LIN {X 0,Y 398.255,Z 601.203,A -85,B 0,C 180,E1 -11633.051,E2 -11633.051} C_VEL
LIN {X 0,Y 399.517,Z 586.027,A -85,B 0,C 180,E1 -11633.934,E2 -11633.934} C_VEL
LIN {X 0,Y 400.58,Z 570.843,A -85,B 0,C 180,E1 -11634.59,E2 -11634.59} C_VEL
LIN {X 0,Y 401.312,Z 556.435,A -85,B 0,C 180,E1 -11635.026,E2 -11635.026} C_VEL
LIN {X 0,Y 404.136,Z 435.509,A -85,B 0,C 180,E1 -11637.319,E2 -11637.319} C_VEL
LIN {X 0,Y 404.064,Z 428.921,A -85,B 0,C 180,E1 -11637.459,E2 -11637.459} C_VEL
LIN {X 0,Y 397.161,Z 389.958,A -85,B 0,C 180,E1 -11638.757,E2 -11638.757} C_VEL
LIN {X 0,Y 397.838,Z 383.514,A -85,B 0,C 180,E1 -11639.811,E2 -11639.811} C_VEL
LIN {X 0,Y 395.942,Z 374.101,A -85,B 0,C 180,E1 -11641.57,E2 -11641.57} C_VEL
LIN {X 0,Y 392.187,Z 359.374,A -85,B 0,C 180,E1 -11644.481,E2 -11644.481} C_VEL
LIN {X 0,Y 390.063,Z 351.524,A -85,B 0,C 180,E1 -11646.11,E2 -11646.11} C_VEL
LIN {X 0,Y 390.067,Z 351.525,A -85,B 0,C 180,E1 -11649.218,E2 -11649.218} C_VEL
LIN {X 0,Y 390.041,Z 351.521,A -85,B 0,C 180,E1 -11652.374,E2 -11652.374} C_VEL
LIN {X 0,Y 390.045,Z 351.526,A -85,B 0,C 180,E1 -11655.355,E2 -11655.355} C_VEL
LIN {X 0,Y 390.029,Z 351.522,A -85,B 0,C 180,E1 -11658.187,E2 -11658.187} C_VEL
LIN {X 0,Y 390.087,Z 351.519,A -85,B 0,C 180,E1 -11660.908,E2 -11660.908} C_VEL
LIN {X 0,Y 390.082,Z 351.519,A -85,B 0,C 180,E1 -11664.793,E2 -11664.793} C_VEL
LIN {X 0,Y 390.02,Z 351.524,A -85,B 0,C 180,E1 -11668.496,E2 -11668.496} C_VEL
LIN {X 0,Y 390.114,Z 351.512,A -85,B 0,C 180,E1 -11672.07,E2 -11672.07} C_VEL
LIN {X 0,Y 390.077,Z 351.519,A -85,B 0,C 180,E1 -11675.519,E2 -11675.519} C_VEL
LIN {X 0,Y 390.052,Z 351.524,A -85,B 0,C 180,E1 -11678.878,E2 -11678.878} C_VEL
LIN {X 0,Y 390.125,Z 351.51,A -85,B 0,C 180,E1 -11682.167,E2 -11682.167} C_VEL
LIN {X 0,Y 390.141,Z 351.511,A -85,B 0,C 180,E1 -11685.393,E2 -11685.393} C_VEL
LIN {X 0,Y 390.145,Z 351.51,A -85,B 0,C 180,E1 -11688.571,E2 -11688.571} C_VEL
LIN {X 0,Y 390.304,Z 351.488,A -85,B 0,C 180,E1 -11692.032,E2 -11692.032} C_VEL
LIN {X 0,Y 390.223,Z 351.504,A -85,B 0,C 180,E1 -11694.834,E2 -11694.834} C_VEL
LIN {X 0,Y 390.418,Z 351.474,A -85,B 0,C 180,E1 -11697.937,E2 -11697.937} C_VEL
LIN {X 0,Y 390.548,Z 351.458,A -85,B 0,C 180,E1 -11700,E2 -11700} C_VEL
LIN {X 0,Y 390.312,Z 351.492,A -85,B 0,C 180,E1 -11703.097,E2 -11703.097} C_VEL
LIN {X 0,Y 390.309,Z 351.487,A -85,B 0,C 180,E1 -11706.612,E2 -11706.612} C_VEL
LIN {X 0,Y 390.203,Z 351.503,A -85,B 0,C 180,E1 -11709.329,E2 -11709.329} C_VEL
LIN {X 0,Y 390.192,Z 351.503,A -85,B 0,C 180,E1 -11713.439,E2 -11713.439} C_VEL
LIN {X 0,Y 390.147,Z 351.509,A -85,B 0,C 180,E1 -11717.308,E2 -11717.308} C_VEL
LIN {X 0,Y 390.085,Z 351.519,A -85,B 0,C 180,E1 -11720.471,E2 -11720.471} C_VEL
LIN {X 0,Y 390.074,Z 351.521,A -85,B 0,C 180,E1 -11724.482,E2 -11724.482} C_VEL
LIN {X 0,Y 390.116,Z 351.512,A -85,B 0,C 180,E1 -11727.931,E2 -11727.931} C_VEL
LIN {X 0,Y 390.022,Z 351.523,A -85,B 0,C 180,E1 -11731.505,E2 -11731.505} C_VEL
LIN {X 0,Y 390.085,Z 351.517,A -85,B 0,C 180,E1 -11735.208,E2 -11735.208} C_VEL
LIN {X 0,Y 390.082,Z 351.518,A -85,B 0,C 180,E1 -11739.094,E2 -11739.094} C_VEL
LIN {X 0,Y 390.038,Z 351.525,A -85,B 0,C 180,E1 -11742.374,E2 -11742.374} C_VEL
LIN {X 0,Y 390.044,Z 351.521,A -85,B 0,C 180,E1 -11745.355,E2 -11745.355} C_VEL
LIN {X 0,Y 390.025,Z 351.526,A -85,B 0,C 180,E1 -11748.187,E2 -11748.187} C_VEL
LIN {X 0,Y 390.083,Z 351.518,A -85,B 0,C 180,E1 -11750.908,E2 -11750.908} C_VEL
LIN {X 0,Y 390.086,Z 351.519,A -85,B 0,C 180,E1 -11754.794,E2 -11754.794} C_VEL
LIN {X 0,Y 390.026,Z 351.53,A -85,B 0,C 180,E1 -11758.496,E2 -11758.496} C_VEL
LIN {X 0,Y 390.04,Z 351.524,A -85,B 0,C 180,E1 -11762.065,E2 -11762.065} C_VEL
LIN {X 0,Y 390.065,Z 351.518,A -85,B 0,C 180,E1 -11765.519,E2 -11765.519} C_VEL
LIN {X 0,Y 390.065,Z 351.52,A -85,B 0,C 180,E1 -11768.879,E2 -11768.879} C_VEL
LIN {X 0,Y 390.092,Z 351.519,A -85,B 0,C 180,E1 -11772.166,E2 -11772.166} C_VEL
LIN {X 0,Y 390.097,Z 351.514,A -85,B 0,C 180,E1 -11775.391,E2 -11775.391} C_VEL
LIN {X 0,Y 390.174,Z 351.504,A -85,B 0,C 180,E1 -11777.518,E2 -11777.518} C_VEL
LIN {X 0,Y 390.195,Z 351.505,A -85,B 0,C 180,E1 -11780.671,E2 -11780.671} C_VEL
LIN {X 0,Y 390.286,Z 351.492,A -85,B 0,C 180,E1 -11783.798,E2 -11783.798} C_VEL
LIN {X 0,Y 390.411,Z 351.478,A -85,B 0,C 180,E1 -11787.937,E2 -11787.937} C_VEL
LIN {X 0,Y 390.41,Z 351.48,A -85,B 0,C 180,E1 -11792.064,E2 -11792.064} C_VEL
LIN {X 0,Y 390.28,Z 351.498,A -85,B 0,C 180,E1 -11796.203,E2 -11796.203} C_VEL
LIN {X 0,Y 390.189,Z 351.502,A -85,B 0,C 180,E1 -11799.33,E2 -11799.33} C_VEL
LIN {X 0,Y 390.153,Z 351.509,A -85,B 0,C 180,E1 -11800.837,E2 -11800.837} C_VEL
LIN {X 0,Y 391.224,Z 354.475,A -85,B 0,C 180,E1 -11801.004,E2 -11801.004} C_VEL
LIN {X 0,Y 399.711,Z 371.741,A -85,B 0,C 180,E1 -11802.004,E2 -11802.004} C_VEL
LIN {X 0,Y 404.687,Z 383.534,A -85,B 0,C 180,E1 -11802.602,E2 -11802.602} C_VEL
LIN {X 0,Y 402.766,Z 468.541,A -85,B 0,C 180,E1 -11804.21,E2 -11804.21} C_VEL
LIN {X 0,Y 402.103,Z 474.385,A -85,B 0,C 180,E1 -11804.286,E2 -11804.286} C_VEL
LIN {X 0,Y 396.37,Z 493.402,A -85,B 0,C 180,E1 -11804.304,E2 -11804.304} C_VEL
LIN {X 0,Y 395.656,Z 499.249,A -85,B 0,C 180,E1 -11804.379,E2 -11804.379} C_VEL
LIN {X 0,Y 395.091,Z 518.571,A -85,B 0,C 180,E1 -11804.816,E2 -11804.816} C_VEL
LIN {X 0,Y 394.423,Z 533.753,A -85,B 0,C 180,E1 -11805.37,E2 -11805.37} C_VEL
LIN {X 0,Y 393.454,Z 548.176,A -85,B 0,C 180,E1 -11806.094,E2 -11806.094} C_VEL
LIN {X 0,Y 392.221,Z 562.984,A -85,B 0,C 180,E1 -11807.063,E2 -11807.063} C_VEL
LIN {X 0,Y 390.965,Z 576.163,A -85,B 0,C 180,E1 -11808.148,E2 -11808.148} C_VEL
LIN {X 0,Y 389.422,Z 589.649,A -85,B 0,C 180,E1 -11809.505,E2 -11809.505} C_VEL
LIN {X 0,Y 388.036,Z 601.503,A -85,B 0,C 180,E1 -11810.96,E2 -11810.96} C_VEL
LIN {X 0,Y 386.753,Z 611.606,A -85,B 0,C 180,E1 -11812.434,E2 -11812.434} C_VEL
LIN {X 0,Y 385.445,Z 622.057,A -85,B 0,C 180,E1 -11814.261,E2 -11814.261} C_VEL
LIN {X 0,Y 384.45,Z 630.439,A -85,B 0,C 180,E1 -11816.024,E2 -11816.024} C_VEL
LIN {X 0,Y 383.572,Z 637.522,A -85,B 0,C 180,E1 -11817.798,E2 -11817.798} C_VEL
LIN {X 0,Y 382.879,Z 643.761,A -85,B 0,C 180,E1 -11819.71,E2 -11819.71} C_VEL
LIN {X 0,Y 382.406,Z 648.694,A -85,B 0,C 180,E1 -11821.587,E2 -11821.587} C_VEL
LIN {X 0,Y 382.038,Z 652.65,A -85,B 0,C 180,E1 -11823.497,E2 -11823.497} C_VEL
LIN {X 0,Y 381.66,Z 656.137,A -85,B 0,C 180,E1 -11825.881,E2 -11825.881} C_VEL
LIN {X 0,Y 381.548,Z 657.743,A -85,B 0,C 180,E1 -11827.622,E2 -11827.622} C_VEL
LIN {X 0,Y 381.509,Z 658.534,A -85,B 0,C 180,E1 -11829.311,E2 -11829.311} C_VEL
LIN {X 0,Y 381.533,Z 658.483,A -85,B 0,C 180,E1 -11831.54,E2 -11831.54} C_VEL
LIN {X 0,Y 381.623,Z 657.767,A -85,B 0,C 180,E1 -11832.953,E2 -11832.953} C_VEL
LIN {X 0,Y 381.786,Z 656.529,A -85,B 0,C 180,E1 -11834.388,E2 -11834.388} C_VEL
LIN {X 0,Y 382.15,Z 653.723,A -85,B 0,C 180,E1 -11836.497,E2 -11836.497} C_VEL
LIN {X 0,Y 382.626,Z 649.129,A -85,B 0,C 180,E1 -11838.859,E2 -11838.859} C_VEL
LIN {X 0,Y 383.213,Z 643.748,A -85,B 0,C 180,E1 -11840.927,E2 -11840.927} C_VEL
LIN {X 0,Y 384.043,Z 637.473,A -85,B 0,C 180,E1 -11842.85,E2 -11842.85} C_VEL
LIN {X 0,Y 385.103,Z 629.901,A -85,B 0,C 180,E1 -11844.745,E2 -11844.745} C_VEL
LIN {X 0,Y 386.331,Z 621.117,A -85,B 0,C 180,E1 -11846.563,E2 -11846.563} C_VEL
LIN {X 0,Y 387.881,Z 610.422,A -85,B 0,C 180,E1 -11848.386,E2 -11848.386} C_VEL
LIN {X 0,Y 389.448,Z 598.829,A -85,B 0,C 180,E1 -11850.022,E2 -11850.022} C_VEL
LIN {X 0,Y 390.945,Z 587.115,A -85,B 0,C 180,E1 -11851.397,E2 -11851.397} C_VEL
LIN {X 0,Y 392.57,Z 573.802,A -85,B 0,C 180,E1 -11852.676,E2 -11852.676} C_VEL
LIN {X 0,Y 393.979,Z 559.343,A -85,B 0,C 180,E1 -11853.8,E2 -11853.8} C_VEL
LIN {X 0,Y 395.149,Z 545.237,A -85,B 0,C 180,E1 -11854.661,E2 -11854.661} C_VEL
LIN {X 0,Y 396.099,Z 530.389,A -85,B 0,C 180,E1 -11855.348,E2 -11855.348} C_VEL
LIN {X 0,Y 396.77,Z 515.087,A -85,B 0,C 180,E1 -11855.842,E2 -11855.842} C_VEL
LIN {X 0,Y 400.24,Z 387.023,A -85,B 0,C 180,E1 -11858.395,E2 -11858.395} C_VEL
LIN {X 0,Y 393.412,Z 372.253,A -85,B 0,C 180,E1 -11859.341,E2 -11859.341} C_VEL
LIN {X 0,Y 386.779,Z 359.714,A -85,B 0,C 180,E1 -11860.28,E2 -11860.28} C_VEL
LIN {X 0,Y 383.378,Z 353.785,A -85,B 0,C 180,E1 -11860.767,E2 -11860.767} C_VEL
LIN {X 0,Y 383.1,Z 352.661,A -85,B 0,C 180,E1 -11860.857,E2 -11860.857} C_VEL
LIN {X 0,Y 383.076,Z 352.389,A -85,B 0,C 180,E1 -11860.995,E2 -11860.995} C_VEL
LIN {X 0,Y 383.024,Z 352.403,A -85,B 0,C 180,E1 -11864.024,E2 -11864.024} C_VEL
LIN {X 0,Y 383.14,Z 352.387,A -85,B 0,C 180,E1 -11867.284,E2 -11867.284} C_VEL
LIN {X 0,Y 383.145,Z 352.383,A -85,B 0,C 180,E1 -11870.497,E2 -11870.497} C_VEL
LIN {X 0,Y 383.237,Z 352.374,A -85,B 0,C 180,E1 -11873.682,E2 -11873.682} C_VEL
LIN {X 0,Y 383.376,Z 352.357,A -85,B 0,C 180,E1 -11877.898,E2 -11877.898} C_VEL
LIN {X 0,Y 383.514,Z 352.338,A -85,B 0,C 180,E1 -11880,E2 -11880} C_VEL
LIN {X 0,Y 383.24,Z 352.372,A -85,B 0,C 180,E1 -11883.153,E2 -11883.153} C_VEL
LIN {X 0,Y 383.245,Z 352.37,A -85,B 0,C 180,E1 -11886.317,E2 -11886.317} C_VEL
LIN {X 0,Y 383.146,Z 352.381,A -85,B 0,C 180,E1 -11889.502,E2 -11889.502} C_VEL
LIN {X 0,Y 383.128,Z 352.384,A -85,B 0,C 180,E1 -11893.536,E2 -11893.536} C_VEL
LIN {X 0,Y 383.096,Z 352.389,A -85,B 0,C 180,E1 -11897.069,E2 -11897.069} C_VEL
LIN {X 0,Y 383.031,Z 352.397,A -85,B 0,C 180,E1 -11900.647,E2 -11900.647} C_VEL
LIN {X 0,Y 383.035,Z 352.393,A -85,B 0,C 180,E1 -11903.807,E2 -11903.807} C_VEL
LIN {X 0,Y 383.082,Z 352.39,A -85,B 0,C 180,E1 -11906.123,E2 -11906.123} C_VEL
LIN {X 0,Y 383.042,Z 352.396,A -85,B 0,C 180,E1 -11908.492,E2 -11908.492} C_VEL
LIN {X 0,Y 383.011,Z 352.397,A -85,B 0,C 180,E1 -11912.149,E2 -11912.149} C_VEL
LIN {X 0,Y 383.019,Z 352.399,A -85,B 0,C 180,E1 -11914.667,E2 -11914.667} C_VEL
LIN {X 0,Y 383.001,Z 352.403,A -85,B 0,C 180,E1 -11917.903,E2 -11917.903} C_VEL
LIN {X 0,Y 382.985,Z 352.404,A -85,B 0,C 180,E1 -11921.347,E2 -11921.347} C_VEL
LIN {X 0,Y 382.998,Z 352.404,A -85,B 0,C 180,E1 -11924.303,E2 -11924.303} C_VEL
LIN {X 0,Y 383.011,Z 352.403,A -85,B 0,C 180,E1 -11927.24,E2 -11927.24} C_VEL
LIN {X 0,Y 383.017,Z 352.4,A -85,B 0,C 180,E1 -11930.413,E2 -11930.413} C_VEL
LIN {X 0,Y 383.024,Z 352.522,A -85,B 0,C 180,E1 -11932.536,E2 -11932.536} C_VEL
LIN {X 0,Y 386.514,Z 364.392,A -85,B 0,C 180,E1 -11935.317,E2 -11935.317} C_VEL
LIN {X 0,Y 389.671,Z 376.604,A -85,B 0,C 180,E1 -11937.96,E2 -11937.96} C_VEL
LIN {X 0,Y 391.472,Z 385.881,A -85,B 0,C 180,E1 -11939.822,E2 -11939.822} C_VEL
LIN {X 0,Y 391.439,Z 387.21,A -85,B 0,C 180,E1 -11940.021,E2 -11940.021} C_VEL
LIN {X 0,Y 396.454,Z 412.815,A -85,B 0,C 180,E1 -11941.057,E2 -11941.057} C_VEL
LIN {X 0,Y 399.417,Z 431.482,A -85,B 0,C 180,E1 -11941.73,E2 -11941.73} C_VEL
LIN {X 0,Y 396.073,Z 554.726,A -85,B 0,C 180,E1 -11944.161,E2 -11944.161} C_VEL
LIN {X 0,Y 395.177,Z 570.565,A -85,B 0,C 180,E1 -11944.663,E2 -11944.663} C_VEL
LIN {X 0,Y 393.997,Z 584.523,A -85,B 0,C 180,E1 -11945.287,E2 -11945.287} C_VEL
LIN {X 0,Y 392.567,Z 598.93,A -85,B 0,C 180,E1 -11946.134,E2 -11946.134} C_VEL
LIN {X 0,Y 391.052,Z 612.302,A -85,B 0,C 180,E1 -11947.129,E2 -11947.129} C_VEL
LIN {X 0,Y 389.444,Z 625.012,A -85,B 0,C 180,E1 -11948.287,E2 -11948.287} C_VEL
LIN {X 0,Y 387.776,Z 637.948,A -85,B 0,C 180,E1 -11949.719,E2 -11949.719} C_VEL
LIN {X 0,Y 386.17,Z 650.24,A -85,B 0,C 180,E1 -11951.366,E2 -11951.366} C_VEL
LIN {X 0,Y 384.888,Z 660.454,A -85,B 0,C 180,E1 -11953.012,E2 -11953.012} C_VEL
LIN {X 0,Y 383.734,Z 670.11,A -85,B 0,C 180,E1 -11954.871,E2 -11954.871} C_VEL
LIN {X 0,Y 382.801,Z 678.511,A -85,B 0,C 180,E1 -11956.82,E2 -11956.82} C_VEL
LIN {X 0,Y 382.269,Z 685.729,A -85,B 0,C 180,E1 -11958.869,E2 -11958.869} C_VEL
LIN {X 0,Y 381.839,Z 691.731,A -85,B 0,C 180,E1 -11960.999,E2 -11960.999} C_VEL
LIN {X 0,Y 381.726,Z 695.327,A -85,B 0,C 180,E1 -11962.595,E2 -11962.595} C_VEL
LIN {X 0,Y 381.649,Z 698.946,A -85,B 0,C 180,E1 -11964.717,E2 -11964.717} C_VEL
LIN {X 0,Y 381.654,Z 701.322,A -85,B 0,C 180,E1 -11966.833,E2 -11966.833} C_VEL
LIN {X 0,Y 381.775,Z 702.066,A -85,B 0,C 180,E1 -11967.89,E2 -11967.89} C_VEL
LIN {X 0,Y 381.723,Z 702.657,A -85,B 0,C 180,E1 -11970,E2 -11970} C_VEL
LIN {X 0,Y 381.775,Z 702.049,A -85,B 0,C 180,E1 -11972.109,E2 -11972.109} C_VEL
LIN {X 0,Y 381.632,Z 700.192,A -85,B 0,C 180,E1 -11974.224,E2 -11974.224} C_VEL
LIN {X 0,Y 381.696,Z 697.121,A -85,B 0,C 180,E1 -11976.342,E2 -11976.342} C_VEL
LIN {X 0,Y 381.791,Z 692.751,A -85,B 0,C 180,E1 -11978.468,E2 -11978.468} C_VEL
LIN {X 0,Y 382.085,Z 686.973,A -85,B 0,C 180,E1 -11980.599,E2 -11980.599} C_VEL
LIN {X 0,Y 382.707,Z 679.641,A -85,B 0,C 180,E1 -11982.73,E2 -11982.73} C_VEL
LIN {X 0,Y 383.471,Z 671.784,A -85,B 0,C 180,E1 -11984.595,E2 -11984.595} C_VEL
LIN {X 0,Y 384.448,Z 662.321,A -85,B 0,C 180,E1 -11986.46,E2 -11986.46} C_VEL
LIN {X 0,Y 385.68,Z 652.713,A -85,B 0,C 180,E1 -11988.045,E2 -11988.045} C_VEL
LIN {X 0,Y 386.954,Z 641.28,A -85,B 0,C 180,E1 -11989.633,E2 -11989.633} C_VEL
LIN {X 0,Y 388.433,Z 628.725,A -85,B 0,C 180,E1 -11991.075,E2 -11991.075} C_VEL
LIN {X 0,Y 390.09,Z 614.856,A -85,B 0,C 180,E1 -11992.37,E2 -11992.37} C_VEL
LIN {X 0,Y 391.633,Z 600.622,A -85,B 0,C 180,E1 -11993.438,E2 -11993.438} C_VEL
LIN {X 0,Y 392.89,Z 586.191,A -85,B 0,C 180,E1 -11994.294,E2 -11994.294} C_VEL
LIN {X 0,Y 393.97,Z 571.213,A -85,B 0,C 180,E1 -11994.96,E2 -11994.96} C_VEL
LIN {X 0,Y 394.801,Z 555.814,A -85,B 0,C 180,E1 -11995.433,E2 -11995.433} C_VEL
LIN {X 0,Y 397.788,Z 432.47,A -85,B 0,C 180,E1 -11997.812,E2 -11997.812} C_VEL
LIN {X 0,Y 397.049,Z 426.368,A -85,B 0,C 180,E1 -11997.992,E2 -11997.992} C_VEL
LIN {X 0,Y 390.521,Z 389.588,A -85,B 0,C 180,E1 -11999.256,E2 -11999.256} C_VEL
LIN {X 0,Y 390.978,Z 385.572,A -85,B 0,C 180,E1 -11999.921,E2 -11999.921} C_VEL
LIN {X 0,Y 390.528,Z 382.108,A -85,B 0,C 180,E1 -12000.556,E2 -12000.556} C_VEL
LIN {X 0,Y 387.141,Z 367.713,A -85,B 0,C 180,E1 -12003.378,E2 -12003.378} C_VEL
LIN {X 0,Y 383.009,Z 352.405,A -85,B 0,C 180,E1 -12006.593,E2 -12006.593} C_VEL
LIN {X 0,Y 383.006,Z 352.398,A -85,B 0,C 180,E1 -12009.958,E2 -12009.958} C_VEL
LIN {X 0,Y 383.002,Z 352.4,A -85,B 0,C 180,E1 -12012.778,E2 -12012.778} C_VEL
LIN {X 0,Y 382.997,Z 352.4,A -85,B 0,C 180,E1 -12015.79,E2 -12015.79} C_VEL
LIN {X 0,Y 382.985,Z 352.402,A -85,B 0,C 180,E1 -12018.796,E2 -12018.796} C_VEL
LIN {X 0,Y 382.998,Z 352.398,A -85,B 0,C 180,E1 -12022.096,E2 -12022.096} C_VEL
LIN {X 0,Y 383.015,Z 352.401,A -85,B 0,C 180,E1 -12025.332,E2 -12025.332} C_VEL
LIN {X 0,Y 382.979,Z 352.407,A -85,B 0,C 180,E1 -12029.081,E2 -12029.081} C_VEL
LIN {X 0,Y 383.053,Z 352.394,A -85,B 0,C 180,E1 -12032.698,E2 -12032.698} C_VEL
LIN {X 0,Y 383.049,Z 352.398,A -85,B 0,C 180,E1 -12035.04,E2 -12035.04} C_VEL
LIN {X 0,Y 382.99,Z 352.4,A -85,B 0,C 180,E1 -12038.469,E2 -12038.469} C_VEL
LIN {X 0,Y 383.06,Z 352.391,A -85,B 0,C 180,E1 -12041.827,E2 -12041.827} C_VEL
LIN {X 0,Y 383.107,Z 352.39,A -85,B 0,C 180,E1 -12045.119,E2 -12045.119} C_VEL
LIN {X 0,Y 383.094,Z 352.387,A -85,B 0,C 180,E1 -12048.358,E2 -12048.358} C_VEL
LIN {X 0,Y 383.26,Z 352.366,A -85,B 0,C 180,E1 -12051.976,E2 -12051.976} C_VEL
LIN {X 0,Y 383.195,Z 352.378,A -85,B 0,C 180,E1 -12054.739,E2 -12054.739} C_VEL
LIN {X 0,Y 383.385,Z 352.35,A -85,B 0,C 180,E1 -12057.899,E2 -12057.899} C_VEL
LIN {X 0,Y 383.517,Z 352.334,A -85,B 0,C 180,E1 -12060,E2 -12060} C_VEL
LIN {X 0,Y 383.248,Z 352.371,A -85,B 0,C 180,E1 -12063.154,E2 -12063.154} C_VEL
LIN {X 0,Y 383.269,Z 352.364,A -85,B 0,C 180,E1 -12066.605,E2 -12066.605} C_VEL
LIN {X 0,Y 383.258,Z 352.368,A -85,B 0,C 180,E1 -12068.436,E2 -12068.436} C_VEL
LIN {X 0,Y 383.095,Z 352.386,A -85,B 0,C 180,E1 -12071.643,E2 -12071.643} C_VEL
LIN {X 0,Y 383.108,Z 352.39,A -85,B 0,C 180,E1 -12074.882,E2 -12074.882} C_VEL
LIN {X 0,Y 383.087,Z 352.388,A -85,B 0,C 180,E1 -12078.173,E2 -12078.173} C_VEL
LIN {X 0,Y 382.99,Z 352.399,A -85,B 0,C 180,E1 -12081.532,E2 -12081.532} C_VEL
LIN {X 0,Y 383.047,Z 352.396,A -85,B 0,C 180,E1 -12084.961,E2 -12084.961} C_VEL
LIN {X 0,Y 383.039,Z 352.398,A -85,B 0,C 180,E1 -12088.493,E2 -12088.493} C_VEL
LIN {X 0,Y 383.008,Z 352.399,A -85,B 0,C 180,E1 -12092.15,E2 -12092.15} C_VEL
LIN {X 0,Y 383.017,Z 352.403,A -85,B 0,C 180,E1 -12094.669,E2 -12094.669} C_VEL
LIN {X 0,Y 382.997,Z 352.399,A -85,B 0,C 180,E1 -12097.904,E2 -12097.904} C_VEL
LIN {X 0,Y 382.98,Z 352.401,A -85,B 0,C 180,E1 -12101.349,E2 -12101.349} C_VEL
LIN {X 0,Y 382.995,Z 352.402,A -85,B 0,C 180,E1 -12104.304,E2 -12104.304} C_VEL
LIN {X 0,Y 383.01,Z 352.397,A -85,B 0,C 180,E1 -12107.241,E2 -12107.241} C_VEL
LIN {X 0,Y 383.005,Z 352.403,A -85,B 0,C 180,E1 -12110.416,E2 -12110.416} C_VEL
LIN {X 0,Y 383.025,Z 352.397,A -85,B 0,C 180,E1 -12114.045,E2 -12114.045} C_VEL
LIN {X 0,Y 382.988,Z 352.399,A -85,B 0,C 180,E1 -12117.579,E2 -12117.579} C_VEL
LIN {X 0,Y 382.982,Z 352.405,A -85,B 0,C 180,E1 -12120.3,E2 -12120.3} C_VEL
LIN {X 0,Y 383.024,Z 352.397,A -85,B 0,C 180,E1 -12124.039,E2 -12124.039} C_VEL
LIN {X 0,Y 383.003,Z 352.398,A -85,B 0,C 180,E1 -12127.335,E2 -12127.335} C_VEL
LIN {X 0,Y 383.045,Z 352.396,A -85,B 0,C 180,E1 -12130.716,E2 -12130.716} C_VEL
LIN {X 0,Y 383.023,Z 352.398,A -85,B 0,C 180,E1 -12134.025,E2 -12134.025} C_VEL
LIN {X 0,Y 383.14,Z 352.381,A -85,B 0,C 180,E1 -12137.285,E2 -12137.285} C_VEL
LIN {X 0,Y 383.146,Z 352.385,A -85,B 0,C 180,E1 -12140.498,E2 -12140.498} C_VEL
LIN {X 0,Y 383.242,Z 352.369,A -85,B 0,C 180,E1 -12143.683,E2 -12143.683} C_VEL
LIN {X 0,Y 383.377,Z 352.354,A -85,B 0,C 180,E1 -12147.899,E2 -12147.899} C_VEL
LIN {X 0,Y 383.376,Z 352.356,A -85,B 0,C 180,E1 -12152.102,E2 -12152.102} C_VEL
LIN {X 0,Y 383.238,Z 352.375,A -85,B 0,C 180,E1 -12156.318,E2 -12156.318} C_VEL
LIN {X 0,Y 383.178,Z 352.38,A -85,B 0,C 180,E1 -12158.438,E2 -12158.438} C_VEL
LIN {X 0,Y 383.123,Z 352.388,A -85,B 0,C 180,E1 -12160.303,E2 -12160.303} C_VEL
LIN {X 0,Y 384.293,Z 355.489,A -85,B 0,C 180,E1 -12160.488,E2 -12160.488} C_VEL
LIN {X 0,Y 393.809,Z 374.728,A -85,B 0,C 180,E1 -12161.638,E2 -12161.638} C_VEL
LIN {X 0,Y 398.39,Z 385.652,A -85,B 0,C 180,E1 -12162.204,E2 -12162.204} C_VEL
LIN {X 0,Y 395.656,Z 499.249,A -85,B 0,C 180,E1 -12164.379,E2 -12164.379} C_VEL
LIN {X 0,Y 394.896,Z 505.096,A -85,B 0,C 180,E1 -12164.451,E2 -12164.451} C_VEL
LIN {X 0,Y 389.314,Z 522.076,A -85,B 0,C 180,E1 -12164.556,E2 -12164.556} C_VEL
LIN {X 0,Y 388.233,Z 527.782,A -85,B 0,C 180,E1 -12164.708,E2 -12164.708} C_VEL
LIN {X 0,Y 388.131,Z 529.686,A -85,B 0,C 180,E1 -12164.779,E2 -12164.779} C_VEL
LIN {X 0,Y 387.175,Z 545.147,A -85,B 0,C 180,E1 -12165.509,E2 -12165.509} C_VEL
LIN {X 0,Y 385.987,Z 559.356,A -85,B 0,C 180,E1 -12166.393,E2 -12166.393} C_VEL
LIN {X 0,Y 384.616,Z 573.623,A -85,B 0,C 180,E1 -12167.523,E2 -12167.523} C_VEL
LIN {X 0,Y 383.028,Z 587.343,A -85,B 0,C 180,E1 -12168.869,E2 -12168.869} C_VEL
LIN {X 0,Y 381.643,Z 598.959,A -85,B 0,C 180,E1 -12170.253,E2 -12170.253} C_VEL
LIN {X 0,Y 380.31,Z 609.104,A -85,B 0,C 180,E1 -12171.691,E2 -12171.691} C_VEL
LIN {X 0,Y 378.93,Z 619.816,A -85,B 0,C 180,E1 -12173.501,E2 -12173.501} C_VEL
LIN {X 0,Y 377.802,Z 628.778,A -85,B 0,C 180,E1 -12175.332,E2 -12175.332} C_VEL
LIN {X 0,Y 376.771,Z 636.38,A -85,B 0,C 180,E1 -12177.194,E2 -12177.194} C_VEL
LIN {X 0,Y 376.005,Z 642.731,A -85,B 0,C 180,E1 -12179.077,E2 -12179.077} C_VEL
LIN {X 0,Y 375.456,Z 648.172,A -85,B 0,C 180,E1 -12181.064,E2 -12181.064} C_VEL
LIN {X 0,Y 375.104,Z 652.153,A -85,B 0,C 180,E1 -12182.912,E2 -12182.912} C_VEL
LIN {X 0,Y 374.799,Z 654.696,A -85,B 0,C 180,E1 -12184.404,E2 -12184.404} C_VEL
LIN {X 0,Y 374.54,Z 656.944,A -85,B 0,C 180,E1 -12186.208,E2 -12186.208} C_VEL
LIN {X 0,Y 374.447,Z 658.532,A -85,B 0,C 180,E1 -12188.271,E2 -12188.271} C_VEL
LIN {X 0,Y 374.422,Z 659.009,A -85,B 0,C 180,E1 -12189.683,E2 -12189.683} C_VEL
LIN {X 0,Y 374.441,Z 658.982,A -85,B 0,C 180,E1 -12191.342,E2 -12191.342} C_VEL
LIN {X 0,Y 374.557,Z 658.236,A -85,B 0,C 180,E1 -12192.964,E2 -12192.964} C_VEL
LIN {X 0,Y 374.731,Z 656.903,A -85,B 0,C 180,E1 -12194.546,E2 -12194.546} C_VEL
LIN {X 0,Y 374.985,Z 655.017,A -85,B 0,C 180,E1 -12196.095,E2 -12196.095} C_VEL
LIN {X 0,Y 375.46,Z 650.83,A -85,B 0,C 180,E1 -12198.482,E2 -12198.482} C_VEL
LIN {X 0,Y 376.051,Z 645.892,A -85,B 0,C 180,E1 -12200.548,E2 -12200.548} C_VEL
LIN {X 0,Y 376.923,Z 639.452,A -85,B 0,C 180,E1 -12202.667,E2 -12202.667} C_VEL
LIN {X 0,Y 378.15,Z 631.111,A -85,B 0,C 180,E1 -12204.861,E2 -12204.861} C_VEL
LIN {X 0,Y 379.451,Z 622.178,A -85,B 0,C 180,E1 -12206.772,E2 -12206.772} C_VEL
LIN {X 0,Y 381.005,Z 612.16,A -85,B 0,C 180,E1 -12208.541,E2 -12208.541} C_VEL
LIN {X 0,Y 382.698,Z 600.337,A -85,B 0,C 180,E1 -12210.275,E2 -12210.275} C_VEL
LIN {X 0,Y 384.364,Z 587.979,A -85,B 0,C 180,E1 -12211.763,E2 -12211.763} C_VEL
LIN {X 0,Y 385.98,Z 575.309,A -85,B 0,C 180,E1 -12213.013,E2 -12213.013} C_VEL
LIN {X 0,Y 387.434,Z 561.584,A -85,B 0,C 180,E1 -12214.119,E2 -12214.119} C_VEL
LIN {X 0,Y 388.72,Z 547.184,A -85,B 0,C 180,E1 -12215.036,E2 -12215.036} C_VEL
LIN {X 0,Y 389.772,Z 531.584,A -85,B 0,C 180,E1 -12215.791,E2 -12215.791} C_VEL
LIN {X 0,Y 390.523,Z 516.021,A -85,B 0,C 180,E1 -12216.309,E2 -12216.309} C_VEL
LIN {X 0,Y 394.22,Z 389.249,A -85,B 0,C 180,E1 -12218.876,E2 -12218.876} C_VEL
LIN {X 0,Y 386.944,Z 373.662,A -85,B 0,C 180,E1 -12219.928,E2 -12219.928} C_VEL
LIN {X 0,Y 381.399,Z 363.396,A -85,B 0,C 180,E1 -12220.734,E2 -12220.734} C_VEL
LIN {X 0,Y 377.736,Z 357.092,A -85,B 0,C 180,E1 -12221.279,E2 -12221.279} C_VEL
LIN {X 0,Y 376.189,Z 354.226,A -85,B 0,C 180,E1 -12221.519,E2 -12221.519} C_VEL
LIN {X 0,Y 376.009,Z 353.297,A -85,B 0,C 180,E1 -12221.585,E2 -12221.585} C_VEL
LIN {X 0,Y 375.994,Z 353.275,A -85,B 0,C 180,E1 -12224.829,E2 -12224.829} C_VEL
LIN {X 0,Y 376.107,Z 353.263,A -85,B 0,C 180,E1 -12227.042,E2 -12227.042} C_VEL
LIN {X 0,Y 376.115,Z 353.26,A -85,B 0,C 180,E1 -12230.318,E2 -12230.318} C_VEL
LIN {X 0,Y 376.196,Z 353.25,A -85,B 0,C 180,E1 -12233.564,E2 -12233.564} C_VEL
LIN {X 0,Y 376.341,Z 353.233,A -85,B 0,C 180,E1 -12237.859,E2 -12237.859} C_VEL
LIN {X 0,Y 376.484,Z 353.213,A -85,B 0,C 180,E1 -12240,E2 -12240} C_VEL
LIN {X 0,Y 376.352,Z 353.227,A -85,B 0,C 180,E1 -12242.14,E2 -12242.14} C_VEL
LIN {X 0,Y 376.203,Z 353.247,A -85,B 0,C 180,E1 -12246.435,E2 -12246.435} C_VEL
LIN {X 0,Y 376.116,Z 353.255,A -85,B 0,C 180,E1 -12249.681,E2 -12249.681} C_VEL
LIN {X 0,Y 376.092,Z 353.261,A -85,B 0,C 180,E1 -12253.657,E2 -12253.657} C_VEL
LIN {X 0,Y 376.035,Z 353.27,A -85,B 0,C 180,E1 -12257.399,E2 -12257.399} C_VEL
LIN {X 0,Y 375.98,Z 353.276,A -85,B 0,C 180,E1 -12260.832,E2 -12260.832} C_VEL
LIN {X 0,Y 375.996,Z 353.269,A -85,B 0,C 180,E1 -12264.281,E2 -12264.281} C_VEL
LIN {X 0,Y 376.022,Z 353.271,A -85,B 0,C 180,E1 -12266.652,E2 -12266.652} C_VEL
LIN {X 0,Y 375.972,Z 353.277,A -85,B 0,C 180,E1 -12269.079,E2 -12269.079} C_VEL
LIN {X 0,Y 375.951,Z 353.278,A -85,B 0,C 180,E1 -12272.828,E2 -12272.828} C_VEL
LIN {X 0,Y 375.959,Z 353.281,A -85,B 0,C 180,E1 -12275.415,E2 -12275.415} C_VEL
LIN {X 0,Y 375.976,Z 353.279,A -85,B 0,C 180,E1 -12278.27,E2 -12278.27} C_VEL
LIN {X 0,Y 375.935,Z 353.283,A -85,B 0,C 180,E1 -12281.6,E2 -12281.6} C_VEL
LIN {X 0,Y 375.955,Z 353.281,A -85,B 0,C 180,E1 -12285.264,E2 -12285.264} C_VEL
LIN {X 0,Y 375.943,Z 353.284,A -85,B 0,C 180,E1 -12289.133,E2 -12289.133} C_VEL
LIN {X 0,Y 375.983,Z 353.406,A -85,B 0,C 180,E1 -12291.869,E2 -12291.869} C_VEL
LIN {X 0,Y 379.799,Z 366.307,A -85,B 0,C 180,E1 -12294.995,E2 -12294.995} C_VEL
LIN {X 0,Y 383.12,Z 379.236,A -85,B 0,C 180,E1 -12297.86,E2 -12297.86} C_VEL
LIN {X 0,Y 384.694,Z 386.664,A -85,B 0,C 180,E1 -12299.361,E2 -12299.361} C_VEL
LIN {X 0,Y 386.24,Z 392.187,A -85,B 0,C 180,E1 -12299.644,E2 -12299.644} C_VEL
LIN {X 0,Y 390.949,Z 417.488,A -85,B 0,C 180,E1 -12300.678,E2 -12300.678} C_VEL
LIN {X 0,Y 393.222,Z 431.966,A -85,B 0,C 180,E1 -12301.209,E2 -12301.209} C_VEL
LIN {X 0,Y 390.249,Z 540.434,A -85,B 0,C 180,E1 -12303.386,E2 -12303.386} C_VEL
LIN {X 0,Y 389.521,Z 558.673,A -85,B 0,C 180,E1 -12303.801,E2 -12303.801} C_VEL
LIN {X 0,Y 388.443,Z 574.566,A -85,B 0,C 180,E1 -12304.371,E2 -12304.371} C_VEL
LIN {X 0,Y 387.106,Z 589.206,A -85,B 0,C 180,E1 -12305.103,E2 -12305.103} C_VEL
LIN {X 0,Y 385.523,Z 603.522,A -85,B 0,C 180,E1 -12306.034,E2 -12306.034} C_VEL
LIN {X 0,Y 383.943,Z 616.674,A -85,B 0,C 180,E1 -12307.109,E2 -12307.109} C_VEL
LIN {X 0,Y 382.152,Z 629.819,A -85,B 0,C 180,E1 -12308.419,E2 -12308.419} C_VEL
LIN {X 0,Y 380.622,Z 640.893,A -85,B 0,C 180,E1 -12309.744,E2 -12309.744} C_VEL
LIN {X 0,Y 379.07,Z 652.626,A -85,B 0,C 180,E1 -12311.43,E2 -12311.43} C_VEL
LIN {X 0,Y 377.606,Z 663.095,A -85,B 0,C 180,E1 -12313.232,E2 -12313.232} C_VEL
LIN {X 0,Y 376.55,Z 672.266,A -85,B 0,C 180,E1 -12315.129,E2 -12315.129} C_VEL
LIN {X 0,Y 375.66,Z 679.915,A -85,B 0,C 180,E1 -12317.026,E2 -12317.026} C_VEL
LIN {X 0,Y 375.057,Z 687.047,A -85,B 0,C 180,E1 -12319.199,E2 -12319.199} C_VEL
LIN {X 0,Y 374.723,Z 692.664,A -85,B 0,C 180,E1 -12321.37,E2 -12321.37} C_VEL
LIN {X 0,Y 374.62,Z 697.502,A -85,B 0,C 180,E1 -12323.877,E2 -12323.877} C_VEL
LIN {X 0,Y 374.559,Z 699.893,A -85,B 0,C 180,E1 -12325.695,E2 -12325.695} C_VEL
LIN {X 0,Y 374.687,Z 701.664,A -85,B 0,C 180,E1 -12327.85,E2 -12327.85} C_VEL
LIN {X 0,Y 374.652,Z 702.243,A -85,B 0,C 180,E1 -12330,E2 -12330} C_VEL
LIN {X 0,Y 374.688,Z 701.628,A -85,B 0,C 180,E1 -12332.149,E2 -12332.149} C_VEL
LIN {X 0,Y 374.557,Z 699.758,A -85,B 0,C 180,E1 -12334.304,E2 -12334.304} C_VEL
LIN {X 0,Y 374.615,Z 696.669,A -85,B 0,C 180,E1 -12336.463,E2 -12336.463} C_VEL
LIN {X 0,Y 374.719,Z 692.277,A -85,B 0,C 180,E1 -12338.629,E2 -12338.629} C_VEL
LIN {X 0,Y 375.055,Z 686.478,A -85,B 0,C 180,E1 -12340.8,E2 -12340.8} C_VEL
LIN {X 0,Y 375.654,Z 679.111,A -85,B 0,C 180,E1 -12342.973,E2 -12342.973} C_VEL
LIN {X 0,Y 376.509,Z 671.219,A -85,B 0,C 180,E1 -12344.871,E2 -12344.871} C_VEL
LIN {X 0,Y 377.556,Z 661.711,A -85,B 0,C 180,E1 -12346.769,E2 -12346.769} C_VEL
LIN {X 0,Y 378.799,Z 652.042,A -85,B 0,C 180,E1 -12348.385,E2 -12348.385} C_VEL
LIN {X 0,Y 380.182,Z 640.544,A -85,B 0,C 180,E1 -12349.998,E2 -12349.998} C_VEL
LIN {X 0,Y 381.757,Z 627.913,A -85,B 0,C 180,E1 -12351.462,E2 -12351.462} C_VEL
LIN {X 0,Y 383.445,Z 613.945,A -85,B 0,C 180,E1 -12352.779,E2 -12352.779} C_VEL
LIN {X 0,Y 385.037,Z 599.957,A -85,B 0,C 180,E1 -12353.837,E2 -12353.837} C_VEL
LIN {X 0,Y 386.365,Z 584.963,A -85,B 0,C 180,E1 -12354.731,E2 -12354.731} C_VEL
LIN {X 0,Y 387.489,Z 569.662,A -85,B 0,C 180,E1 -12355.407,E2 -12355.407} C_VEL
LIN {X 0,Y 388.314,Z 555.039,A -85,B 0,C 180,E1 -12355.853,E2 -12355.853} C_VEL
LIN {X 0,Y 391.382,Z 433.252,A -85,B 0,C 180,E1 -12358.243,E2 -12358.243} C_VEL
LIN {X 0,Y 390.29,Z 425.225,A -85,B 0,C 180,E1 -12358.495,E2 -12358.495} C_VEL
LIN {X 0,Y 383.901,Z 389.155,A -85,B 0,C 180,E1 -12359.774,E2 -12359.774} C_VEL
LIN {X 0,Y 384.095,Z 385.641,A -85,B 0,C 180,E1 -12360.384,E2 -12360.384} C_VEL
LIN {X 0,Y 380.797,Z 371.444,A -85,B 0,C 180,E1 -12363.199,E2 -12363.199} C_VEL
LIN {X 0,Y 376.51,Z 355.246,A -85,B 0,C 180,E1 -12366.617,E2 -12366.617} C_VEL
LIN {X 0,Y 375.957,Z 353.282,A -85,B 0,C 180,E1 -12367.075,E2 -12367.075} C_VEL
LIN {X 0,Y 375.986,Z 353.272,A -85,B 0,C 180,E1 -12369.97,E2 -12369.97} C_VEL
LIN {X 0,Y 375.929,Z 353.28,A -85,B 0,C 180,E1 -12373.765,E2 -12373.765} C_VEL
LIN {X 0,Y 375.931,Z 353.281,A -85,B 0,C 180,E1 -12376.81,E2 -12376.81} C_VEL
LIN {X 0,Y 375.959,Z 353.276,A -85,B 0,C 180,E1 -12380.537,E2 -12380.537} C_VEL
LIN {X 0,Y 375.961,Z 353.278,A -85,B 0,C 180,E1 -12383.495,E2 -12383.495} C_VEL
LIN {X 0,Y 375.956,Z 353.276,A -85,B 0,C 180,E1 -12385.889,E2 -12385.889} C_VEL
LIN {X 0,Y 375.961,Z 353.276,A -85,B 0,C 180,E1 -12389.687,E2 -12389.687} C_VEL
LIN {X 0,Y 375.992,Z 353.271,A -85,B 0,C 180,E1 -12392.141,E2 -12392.141} C_VEL
LIN {X 0,Y 376.003,Z 353.271,A -85,B 0,C 180,E1 -12394.539,E2 -12394.539} C_VEL
LIN {X 0,Y 375.96,Z 353.275,A -85,B 0,C 180,E1 -12398.046,E2 -12398.046} C_VEL
LIN {X 0,Y 376.006,Z 353.271,A -85,B 0,C 180,E1 -12401.473,E2 -12401.473} C_VEL
LIN {X 0,Y 376.055,Z 353.268,A -85,B 0,C 180,E1 -12404.833,E2 -12404.833} C_VEL
LIN {X 0,Y 376.047,Z 353.264,A -85,B 0,C 180,E1 -12408.137,E2 -12408.137} C_VEL
LIN {X 0,Y 376.215,Z 353.243,A -85,B 0,C 180,E1 -12411.919,E2 -12411.919} C_VEL
LIN {X 0,Y 376.167,Z 353.253,A -85,B 0,C 180,E1 -12414.64,E2 -12414.64} C_VEL
LIN {X 0,Y 376.351,Z 353.226,A -85,B 0,C 180,E1 -12417.86,E2 -12417.86} C_VEL
LIN {X 0,Y 376.486,Z 353.209,A -85,B 0,C 180,E1 -12420,E2 -12420} C_VEL
LIN {X 0,Y 376.186,Z 353.25,A -85,B 0,C 180,E1 -12423.213,E2 -12423.213} C_VEL
LIN {X 0,Y 376.234,Z 353.242,A -85,B 0,C 180,E1 -12426.596,E2 -12426.596} C_VEL
LIN {X 0,Y 376.203,Z 353.249,A -85,B 0,C 180,E1 -12428.596,E2 -12428.596} C_VEL
LIN {X 0,Y 376.048,Z 353.264,A -85,B 0,C 180,E1 -12431.864,E2 -12431.864} C_VEL
LIN {X 0,Y 376.056,Z 353.266,A -85,B 0,C 180,E1 -12435.168,E2 -12435.168} C_VEL
LIN {X 0,Y 376.022,Z 353.271,A -85,B 0,C 180,E1 -12438.527,E2 -12438.527} C_VEL
LIN {X 0,Y 375.955,Z 353.276,A -85,B 0,C 180,E1 -12441.955,E2 -12441.955} C_VEL
LIN {X 0,Y 376.003,Z 353.27,A -85,B 0,C 180,E1 -12445.462,E2 -12445.462} C_VEL
LIN {X 0,Y 375.969,Z 353.276,A -85,B 0,C 180,E1 -12449.08,E2 -12449.08} C_VEL
LIN {X 0,Y 375.948,Z 353.281,A -85,B 0,C 180,E1 -12452.829,E2 -12452.829} C_VEL
LIN {X 0,Y 375.957,Z 353.276,A -85,B 0,C 180,E1 -12455.416,E2 -12455.416} C_VEL
LIN {X 0,Y 375.97,Z 353.277,A -85,B 0,C 180,E1 -12458.271,E2 -12458.271} C_VEL
LIN {X 0,Y 375.932,Z 353.278,A -85,B 0,C 180,E1 -12461.601,E2 -12461.601} C_VEL
LIN {X 0,Y 375.926,Z 353.28,A -85,B 0,C 180,E1 -12465.269,E2 -12465.269} C_VEL
LIN {X 0,Y 375.924,Z 353.284,A -85,B 0,C 180,E1 -12468.402,E2 -12468.402} C_VEL
LIN {X 0,Y 375.971,Z 353.274,A -85,B 0,C 180,E1 -12471.731,E2 -12471.731} C_VEL
LIN {X 0,Y 375.981,Z 353.273,A -85,B 0,C 180,E1 -12475.333,E2 -12475.333} C_VEL
LIN {X 0,Y 375.959,Z 353.281,A -85,B 0,C 180,E1 -12478.439,E2 -12478.439} C_VEL
LIN {X 0,Y 375.936,Z 353.281,A -85,B 0,C 180,E1 -12482.137,E2 -12482.137} C_VEL
LIN {X 0,Y 375.982,Z 353.273,A -85,B 0,C 180,E1 -12485.718,E2 -12485.718} C_VEL
LIN {X 0,Y 376.001,Z 353.27,A -85,B 0,C 180,E1 -12489.199,E2 -12489.199} C_VEL
LIN {X 0,Y 376.013,Z 353.273,A -85,B 0,C 180,E1 -12492.6,E2 -12492.6} C_VEL
LIN {X 0,Y 376.093,Z 353.265,A -85,B 0,C 180,E1 -12496.343,E2 -12496.343} C_VEL
LIN {X 0,Y 376.116,Z 353.262,A -85,B 0,C 180,E1 -12500.319,E2 -12500.319} C_VEL
LIN {X 0,Y 376.201,Z 353.245,A -85,B 0,C 180,E1 -12503.565,E2 -12503.565} C_VEL
LIN {X 0,Y 376.342,Z 353.23,A -85,B 0,C 180,E1 -12507.86,E2 -12507.86} C_VEL
LIN {X 0,Y 376.341,Z 353.233,A -85,B 0,C 180,E1 -12512.141,E2 -12512.141} C_VEL
LIN {X 0,Y 376.198,Z 353.251,A -85,B 0,C 180,E1 -12516.436,E2 -12516.436} C_VEL
LIN {X 0,Y 376.139,Z 353.255,A -85,B 0,C 180,E1 -12518.597,E2 -12518.597} C_VEL
LIN {X 0,Y 376.094,Z 353.26,A -85,B 0,C 180,E1 -12519.75,E2 -12519.75} C_VEL
LIN {X 0,Y 377.11,Z 356.135,A -85,B 0,C 180,E1 -12519.924,E2 -12519.924} C_VEL
LIN {X 0,Y 387.616,Z 377.08,A -85,B 0,C 180,E1 -12521.223,E2 -12521.223} C_VEL
LIN {X 0,Y 392.036,Z 387.774,A -85,B 0,C 180,E1 -12521.789,E2 -12521.789} C_VEL
LIN {X 0,Y 388.796,Z 514.884,A -85,B 0,C 180,E1 -12524.292,E2 -12524.292} C_VEL
LIN {X 0,Y 388.131,Z 529.686,A -85,B 0,C 180,E1 -12524.779,E2 -12524.779} C_VEL
LIN {X 0,Y 387.347,Z 535.365,A -85,B 0,C 180,E1 -12524.983,E2 -12524.983} C_VEL
LIN {X 0,Y 384.095,Z 544.524,A -85,B 0,C 180,E1 -12525.271,E2 -12525.271} C_VEL
LIN {X 0,Y 380.614,Z 553.583,A -85,B 0,C 180,E1 -12525.631,E2 -12525.631} C_VEL
LIN {X 0,Y 379.475,Z 558.92,A -85,B 0,C 180,E1 -12525.948,E2 -12525.948} C_VEL
LIN {X 0,Y 378.169,Z 572.494,A -85,B 0,C 180,E1 -12527.02,E2 -12527.02} C_VEL
LIN {X 0,Y 376.541,Z 586.126,A -85,B 0,C 180,E1 -12528.342,E2 -12528.342} C_VEL
LIN {X 0,Y 374.952,Z 598.735,A -85,B 0,C 180,E1 -12529.844,E2 -12529.844} C_VEL
LIN {X 0,Y 373.382,Z 610.442,A -85,B 0,C 180,E1 -12531.534,E2 -12531.534} C_VEL
LIN {X 0,Y 371.963,Z 620.997,A -85,B 0,C 180,E1 -12533.378,E2 -12533.378} C_VEL
LIN {X 0,Y 370.803,Z 629.849,A -85,B 0,C 180,E1 -12535.243,E2 -12535.243} C_VEL
LIN {X 0,Y 369.724,Z 637.348,A -85,B 0,C 180,E1 -12537.143,E2 -12537.143} C_VEL
LIN {X 0,Y 368.889,Z 644.064,A -85,B 0,C 180,E1 -12539.222,E2 -12539.222} C_VEL
LIN {X 0,Y 368.39,Z 648.744,A -85,B 0,C 180,E1 -12541.004,E2 -12541.004} C_VEL
LIN {X 0,Y 368.05,Z 652.608,A -85,B 0,C 180,E1 -12542.839,E2 -12542.839} C_VEL
LIN {X 0,Y 367.601,Z 656,A -85,B 0,C 180,E1 -12544.999,E2 -12544.999} C_VEL
LIN {X 0,Y 367.436,Z 657.751,A -85,B 0,C 180,E1 -12546.549,E2 -12546.549} C_VEL
LIN {X 0,Y 367.354,Z 658.972,A -85,B 0,C 180,E1 -12548.335,E2 -12548.335} C_VEL
LIN {X 0,Y 367.337,Z 659.485,A -85,B 0,C 180,E1 -12550.58,E2 -12550.58} C_VEL
LIN {X 0,Y 367.389,Z 659.165,A -85,B 0,C 180,E1 -12552.032,E2 -12552.032} C_VEL
LIN {X 0,Y 367.525,Z 658.342,A -85,B 0,C 180,E1 -12553.505,E2 -12553.505} C_VEL
LIN {X 0,Y 367.839,Z 656.047,A -85,B 0,C 180,E1 -12555.765,E2 -12555.765} C_VEL
LIN {X 0,Y 368.287,Z 652.353,A -85,B 0,C 180,E1 -12558.094,E2 -12558.094} C_VEL
LIN {X 0,Y 368.938,Z 647.31,A -85,B 0,C 180,E1 -12560.386,E2 -12560.386} C_VEL
LIN {X 0,Y 369.808,Z 641.16,A -85,B 0,C 180,E1 -12562.544,E2 -12562.544} C_VEL
LIN {X 0,Y 370.933,Z 634.004,A -85,B 0,C 180,E1 -12564.56,E2 -12564.56} C_VEL
LIN {X 0,Y 372.22,Z 625.519,A -85,B 0,C 180,E1 -12566.523,E2 -12566.523} C_VEL
LIN {X 0,Y 373.841,Z 615.671,A -85,B 0,C 180,E1 -12568.396,E2 -12568.396} C_VEL
LIN {X 0,Y 375.519,Z 604.799,A -85,B 0,C 180,E1 -12570.112,E2 -12570.112} C_VEL
LIN {X 0,Y 377.141,Z 593.279,A -85,B 0,C 180,E1 -12571.628,E2 -12571.628} C_VEL
LIN {X 0,Y 378.969,Z 579.904,A -85,B 0,C 180,E1 -12573.07,E2 -12573.07} C_VEL
LIN {X 0,Y 380.576,Z 566.902,A -85,B 0,C 180,E1 -12574.211,E2 -12574.211} C_VEL
LIN {X 0,Y 381.919,Z 553.315,A -85,B 0,C 180,E1 -12575.178,E2 -12575.178} C_VEL
LIN {X 0,Y 383.108,Z 538.751,A -85,B 0,C 180,E1 -12575.982,E2 -12575.982} C_VEL
LIN {X 0,Y 383.991,Z 524.057,A -85,B 0,C 180,E1 -12576.579,E2 -12576.579} C_VEL
LIN {X 0,Y 384.594,Z 508.64,A -85,B 0,C 180,E1 -12576.991,E2 -12576.991} C_VEL
LIN {X 0,Y 388.074,Z 391.123,A -85,B 0,C 180,E1 -12579.402,E2 -12579.402} C_VEL
LIN {X 0,Y 380.44,Z 375.036,A -85,B 0,C 180,E1 -12580.543,E2 -12580.543} C_VEL
LIN {X 0,Y 373.014,Z 361.748,A -85,B 0,C 180,E1 -12581.674,E2 -12581.674} C_VEL
LIN {X 0,Y 370.487,Z 357.684,A -85,B 0,C 180,E1 -12582.066,E2 -12582.066} C_VEL
LIN {X 0,Y 369.256,Z 355.345,A -85,B 0,C 180,E1 -12582.27,E2 -12582.27} C_VEL
LIN {X 0,Y 369,Z 354.142,A -85,B 0,C 180,E1 -12582.358,E2 -12582.358} C_VEL
LIN {X 0,Y 369.061,Z 354.14,A -85,B 0,C 180,E1 -12586.79,E2 -12586.79} C_VEL
LIN {X 0,Y 369.066,Z 354.139,A -85,B 0,C 180,E1 -12590.131,E2 -12590.131} C_VEL
LIN {X 0,Y 369.158,Z 354.126,A -85,B 0,C 180,E1 -12593.441,E2 -12593.441} C_VEL
LIN {X 0,Y 369.305,Z 354.108,A -85,B 0,C 180,E1 -12597.818,E2 -12597.818} C_VEL
LIN {X 0,Y 369.433,Z 354.091,A -85,B 0,C 180,E1 -12600,E2 -12600} C_VEL
LIN {X 0,Y 369.316,Z 354.103,A -85,B 0,C 180,E1 -12602.181,E2 -12602.181} C_VEL
LIN {X 0,Y 369.163,Z 354.124,A -85,B 0,C 180,E1 -12606.559,E2 -12606.559} C_VEL
LIN {X 0,Y 369.066,Z 354.133,A -85,B 0,C 180,E1 -12609.868,E2 -12609.868} C_VEL
LIN {X 0,Y 369.04,Z 354.14,A -85,B 0,C 180,E1 -12613.772,E2 -12613.772} C_VEL
LIN {X 0,Y 368.993,Z 354.144,A -85,B 0,C 180,E1 -12617.742,E2 -12617.742} C_VEL
LIN {X 0,Y 368.931,Z 354.151,A -85,B 0,C 180,E1 -12621.219,E2 -12621.219} C_VEL
LIN {X 0,Y 368.96,Z 354.146,A -85,B 0,C 180,E1 -12624.775,E2 -12624.775} C_VEL
LIN {X 0,Y 368.97,Z 354.146,A -85,B 0,C 180,E1 -12627.203,E2 -12627.203} C_VEL
LIN {X 0,Y 368.921,Z 354.152,A -85,B 0,C 180,E1 -12629.689,E2 -12629.689} C_VEL
LIN {X 0,Y 368.898,Z 354.158,A -85,B 0,C 180,E1 -12633.043,E2 -12633.043} C_VEL
LIN {X 0,Y 368.919,Z 354.157,A -85,B 0,C 180,E1 -12636.196,E2 -12636.196} C_VEL
LIN {X 0,Y 368.905,Z 354.158,A -85,B 0,C 180,E1 -12638.953,E2 -12638.953} C_VEL
LIN {X 0,Y 368.882,Z 354.162,A -85,B 0,C 180,E1 -12642.009,E2 -12642.009} C_VEL
LIN {X 0,Y 368.928,Z 354.156,A -85,B 0,C 180,E1 -12645.183,E2 -12645.183} C_VEL
LIN {X 0,Y 368.885,Z 354.162,A -85,B 0,C 180,E1 -12648.177,E2 -12648.177} C_VEL
LIN {X 0,Y 368.921,Z 354.221,A -85,B 0,C 180,E1 -12651.149,E2 -12651.149} C_VEL
LIN {X 0,Y 372.622,Z 366.344,A -85,B 0,C 180,E1 -12654.219,E2 -12654.219} C_VEL
LIN {X 0,Y 375.5,Z 377.574,A -85,B 0,C 180,E1 -12656.807,E2 -12656.807} C_VEL
LIN {X 0,Y 377.426,Z 385.926,A -85,B 0,C 180,E1 -12658.609,E2 -12658.609} C_VEL
LIN {X 0,Y 379.943,Z 392.127,A -85,B 0,C 180,E1 -12659.023,E2 -12659.023} C_VEL
LIN {X 0,Y 384.71,Z 417.394,A -85,B 0,C 180,E1 -12660.1,E2 -12660.1} C_VEL
LIN {X 0,Y 387.163,Z 433.623,A -85,B 0,C 180,E1 -12660.711,E2 -12660.711} C_VEL
LIN {X 0,Y 383.519,Z 554.01,A -85,B 0,C 180,E1 -12663.175,E2 -12663.175} C_VEL
LIN {X 0,Y 382.54,Z 569.697,A -85,B 0,C 180,E1 -12663.69,E2 -12663.69} C_VEL
LIN {X 0,Y 381.147,Z 584.84,A -85,B 0,C 180,E1 -12664.394,E2 -12664.394} C_VEL
LIN {X 0,Y 379.539,Z 599.554,A -85,B 0,C 180,E1 -12665.308,E2 -12665.308} C_VEL
LIN {X 0,Y 377.764,Z 613.675,A -85,B 0,C 180,E1 -12666.422,E2 -12666.422} C_VEL
LIN {X 0,Y 375.869,Z 627.266,A -85,B 0,C 180,E1 -12667.75,E2 -12667.75} C_VEL
LIN {X 0,Y 374.052,Z 639.682,A -85,B 0,C 180,E1 -12669.228,E2 -12669.228} C_VEL
LIN {X 0,Y 372.287,Z 651.904,A -85,B 0,C 180,E1 -12670.998,E2 -12670.998} C_VEL
LIN {X 0,Y 370.965,Z 661.401,A -85,B 0,C 180,E1 -12672.639,E2 -12672.639} C_VEL
LIN {X 0,Y 369.706,Z 670.744,A -85,B 0,C 180,E1 -12674.565,E2 -12674.565} C_VEL
LIN {X 0,Y 368.835,Z 677.997,A -85,B 0,C 180,E1 -12676.356,E2 -12676.356} C_VEL
LIN {X 0,Y 368.179,Z 685.022,A -85,B 0,C 180,E1 -12678.437,E2 -12678.437} C_VEL
LIN {X 0,Y 367.711,Z 691.001,A -85,B 0,C 180,E1 -12680.65,E2 -12680.65} C_VEL
LIN {X 0,Y 367.567,Z 694.586,A -85,B 0,C 180,E1 -12682.308,E2 -12682.308} C_VEL
LIN {X 0,Y 367.476,Z 698.178,A -85,B 0,C 180,E1 -12684.512,E2 -12684.512} C_VEL
LIN {X 0,Y 367.467,Z 700.529,A -85,B 0,C 180,E1 -12686.71,E2 -12686.71} C_VEL
LIN {X 0,Y 367.594,Z 701.692,A -85,B 0,C 180,E1 -12688.904,E2 -12688.904} C_VEL
LIN {X 0,Y 367.594,Z 701.669,A -85,B 0,C 180,E1 -12691.095,E2 -12691.095} C_VEL
LIN {X 0,Y 367.603,Z 701.203,A -85,B 0,C 180,E1 -12692.191,E2 -12692.191} C_VEL
LIN {X 0,Y 367.483,Z 699.317,A -85,B 0,C 180,E1 -12694.387,E2 -12694.387} C_VEL
LIN {X 0,Y 367.544,Z 696.206,A -85,B 0,C 180,E1 -12696.588,E2 -12696.588} C_VEL
LIN {X 0,Y 367.635,Z 691.786,A -85,B 0,C 180,E1 -12698.797,E2 -12698.797} C_VEL
LIN {X 0,Y 368.027,Z 685.957,A -85,B 0,C 180,E1 -12701.009,E2 -12701.009} C_VEL
LIN {X 0,Y 368.582,Z 679.588,A -85,B 0,C 180,E1 -12702.946,E2 -12702.946} C_VEL
LIN {X 0,Y 369.414,Z 671.883,A -85,B 0,C 180,E1 -12704.882,E2 -12704.882} C_VEL
LIN {X 0,Y 370.472,Z 662.589,A -85,B 0,C 180,E1 -12706.815,E2 -12706.815} C_VEL
LIN {X 0,Y 371.774,Z 653.104,A -85,B 0,C 180,E1 -12708.459,E2 -12708.459} C_VEL
LIN {X 0,Y 373.147,Z 641.869,A -85,B 0,C 180,E1 -12710.104,E2 -12710.104} C_VEL
LIN {X 0,Y 374.7,Z 629.58,A -85,B 0,C 180,E1 -12711.598,E2 -12711.598} C_VEL
LIN {X 0,Y 376.453,Z 616.11,A -85,B 0,C 180,E1 -12712.936,E2 -12712.936} C_VEL
LIN {X 0,Y 378.069,Z 602.945,A -85,B 0,C 180,E1 -12713.993,E2 -12713.993} C_VEL
LIN {X 0,Y 379.445,Z 588.673,A -85,B 0,C 180,E1 -12714.916,E2 -12714.916} C_VEL
LIN {X 0,Y 380.659,Z 573.949,A -85,B 0,C 180,E1 -12715.64,E2 -12715.64} C_VEL
LIN {X 0,Y 381.594,Z 559.119,A -85,B 0,C 180,E1 -12716.159,E2 -12716.159} C_VEL
LIN {X 0,Y 382.343,Z 538.185,A -85,B 0,C 180,E1 -12716.618,E2 -12716.618} C_VEL
LIN {X 0,Y 384.987,Z 434.063,A -85,B 0,C 180,E1 -12718.689,E2 -12718.689} C_VEL
LIN {X 0,Y 384.085,Z 427.329,A -85,B 0,C 180,E1 -12718.904,E2 -12718.904} C_VEL
LIN {X 0,Y 377.339,Z 388.778,A -85,B 0,C 180,E1 -12720.302,E2 -12720.302} C_VEL
LIN {X 0,Y 376.201,Z 382.422,A -85,B 0,C 180,E1 -12721.539,E2 -12721.539} C_VEL
LIN {X 0,Y 372.761,Z 368.339,A -85,B 0,C 180,E1 -12724.444,E2 -12724.444} C_VEL
LIN {X 0,Y 368.928,Z 354.158,A -85,B 0,C 180,E1 -12727.559,E2 -12727.559} C_VEL
LIN {X 0,Y 368.908,Z 354.154,A -85,B 0,C 180,E1 -12730.37,E2 -12730.37} C_VEL
LIN {X 0,Y 368.882,Z 354.159,A -85,B 0,C 180,E1 -12733.616,E2 -12733.616} C_VEL
LIN {X 0,Y 368.883,Z 354.158,A -85,B 0,C 180,E1 -12736.696,E2 -12736.696} C_VEL
LIN {X 0,Y 368.908,Z 354.155,A -85,B 0,C 180,E1 -12739.643,E2 -12739.643} C_VEL
LIN {X 0,Y 368.899,Z 354.161,A -85,B 0,C 180,E1 -12743.144,E2 -12743.144} C_VEL
LIN {X 0,Y 368.893,Z 354.156,A -85,B 0,C 180,E1 -12746.462,E2 -12746.462} C_VEL
LIN {X 0,Y 368.925,Z 354.157,A -85,B 0,C 180,E1 -12749.046,E2 -12749.046} C_VEL
LIN {X 0,Y 368.976,Z 354.147,A -85,B 0,C 180,E1 -12751.564,E2 -12751.564} C_VEL
LIN {X 0,Y 368.996,Z 354.142,A -85,B 0,C 180,E1 -12754.02,E2 -12754.02} C_VEL
LIN {X 0,Y 368.929,Z 354.152,A -85,B 0,C 180,E1 -12757.605,E2 -12757.605} C_VEL
LIN {X 0,Y 368.955,Z 354.154,A -85,B 0,C 180,E1 -12761.106,E2 -12761.106} C_VEL
LIN {X 0,Y 368.995,Z 354.145,A -85,B 0,C 180,E1 -12764.535,E2 -12764.535} C_VEL
LIN {X 0,Y 369.002,Z 354.142,A -85,B 0,C 180,E1 -12767.907,E2 -12767.907} C_VEL
LIN {X 0,Y 369.184,Z 354.119,A -85,B 0,C 180,E1 -12771.846,E2 -12771.846} C_VEL
LIN {X 0,Y 369.139,Z 354.127,A -85,B 0,C 180,E1 -12774.538,E2 -12774.538} C_VEL
LIN {X 0,Y 369.316,Z 354.103,A -85,B 0,C 180,E1 -12777.819,E2 -12777.819} C_VEL
LIN {X 0,Y 369.456,Z 354.085,A -85,B 0,C 180,E1 -12780,E2 -12780} C_VEL
LIN {X 0,Y 369.316,Z 354.103,A -85,B 0,C 180,E1 -12782.182,E2 -12782.182} C_VEL
LIN {X 0,Y 369.205,Z 354.12,A -85,B 0,C 180,E1 -12786.583,E2 -12786.583} C_VEL
LIN {X 0,Y 369.136,Z 354.131,A -85,B 0,C 180,E1 -12788.761,E2 -12788.761} C_VEL
LIN {X 0,Y 369.003,Z 354.142,A -85,B 0,C 180,E1 -12792.094,E2 -12792.094} C_VEL
LIN {X 0,Y 368.996,Z 354.143,A -85,B 0,C 180,E1 -12795.465,E2 -12795.465} C_VEL
LIN {X 0,Y 368.981,Z 354.15,A -85,B 0,C 180,E1 -12798.893,E2 -12798.893} C_VEL
LIN {X 0,Y 368.921,Z 354.155,A -85,B 0,C 180,E1 -12802.396,E2 -12802.396} C_VEL
LIN {X 0,Y 368.997,Z 354.143,A -85,B 0,C 180,E1 -12805.981,E2 -12805.981} C_VEL
LIN {X 0,Y 368.96,Z 354.152,A -85,B 0,C 180,E1 -12808.812,E2 -12808.812} C_VEL
LIN {X 0,Y 368.897,Z 354.157,A -85,B 0,C 180,E1 -12812.239,E2 -12812.239} C_VEL
LIN {X 0,Y 368.928,Z 354.154,A -85,B 0,C 180,E1 -12815.002,E2 -12815.002} C_VEL
LIN {X 0,Y 368.905,Z 354.161,A -85,B 0,C 180,E1 -12818.64,E2 -12818.64} C_VEL
LIN {X 0,Y 368.879,Z 354.158,A -85,B 0,C 180,E1 -12822.01,E2 -12822.01} C_VEL
LIN {X 0,Y 368.879,Z 354.158,A -85,B 0,C 180,E1 -12825.176,E2 -12825.176} C_VEL
LIN {X 0,Y 368.875,Z 354.16,A -85,B 0,C 180,E1 -12828.177,E2 -12828.177} C_VEL
LIN {X 0,Y 368.903,Z 354.154,A -85,B 0,C 180,E1 -12831.362,E2 -12831.362} C_VEL
LIN {X 0,Y 368.937,Z 354.151,A -85,B 0,C 180,E1 -12835.147,E2 -12835.147} C_VEL
LIN {X 0,Y 368.931,Z 354.152,A -85,B 0,C 180,E1 -12839.047,E2 -12839.047} C_VEL
LIN {X 0,Y 368.879,Z 354.16,A -85,B 0,C 180,E1 -12842.79,E2 -12842.79} C_VEL
LIN {X 0,Y 368.935,Z 354.153,A -85,B 0,C 180,E1 -12846.118,E2 -12846.118} C_VEL
LIN {X 0,Y 368.932,Z 354.152,A -85,B 0,C 180,E1 -12849.947,E2 -12849.947} C_VEL
LIN {X 0,Y 368.929,Z 354.151,A -85,B 0,C 180,E1 -12853.397,E2 -12853.397} C_VEL
